# B&R Automation Studio project A2019059_Linka_Power_CP (part 19)

```iecst
            IF NOT SC_P1_Srobovanie.Switch2 AND SC_OvlManipulatora_OsY.Step = 1 AND P1_Srobovacky_VychodziaPozicia AND P1_Srobovanie.STAV.OsX_PoziciaDosiahnuta AND Safety.STAV.P1_ZonaBunky_AKTIVNA THEN
                OsY_POLOHUJ:= TRUE;
                SC_P1_Srobovanie.Switch2:= TRUE;
            END_IF

            IF P1_Srobovanie.STAV.OsX_PoziciaDosiahnuta AND P1_Srobovanie.STAV.OsY_PoziciaDosiahnuta THEN
                P1_Srobovanie.STAV.OsX_PoziciaDosiahnuta:= FALSE;
                P1_Srobovanie.STAV.OsY_PoziciaDosiahnuta:= FALSE;
                SC_P1_Srobovanie.ResetStep:= TRUE;
                SC_P1_Srobovanie.Step:= 503;
            END_IF

        503:
            SC_P1_Srobovanie.StepName:='503 - Inicializacia - zahodenie skrutky K30';
            SC_P1_Srobovanie.IdleTime.PT:= T#30s;
            SC_P1_Srobovanie.AlarmTime.PT:= T#30s;
            SC_P1_Srobovanie.IdleTime.IN:= TRUE;

            IF NOT SC_P1_Srobovanie.Switch1 THEN
                P1_Srobovanie.SkrutkovaciSet_K30.Cistenie:= TRUE;
                SC_P1_Srobovanie.Switch1:= TRUE;
            END_IF

            IF P1_Srobovanie.SkrutkovaciSet_K30.CistenieUkoncene AND P1_Srobovanie.IN.SkrutkK30_ZASUNUTY_MS20 THEN
                P1_Srobovanie.SkrutkovaciSet_K30.Cistenie:= FALSE;
            END_IF

            IF NOT P1_Srobovanie.SkrutkovaciSet_K30.Cistenie AND P1_Srobovanie.SkrutkovaciSet_K30.SkrutkaK30_Pripravena AND SC_P1_Srobovanie.Switch1 THEN
                P1_Srobovanie.STAV.Cistenie_K30_BUSY:= FALSE;
                P1_Srobovanie.RR_SkrutkovackaK30_CISTENIE:= FALSE;
                SC_P1_Srobovanie.ResetStep:= TRUE;
                SC_P1_Srobovanie.Step:= FazaNavratu;
            ELSIF SC_P1_Srobovanie.IdleTime.Q THEN
                SC_P1_Srobovanie.ResetStep:= TRUE;
                SC_P1_Srobovanie.Step:= 505;
            END_IF

        505:
            SC_P1_Srobovanie.StepName:='505 - Inicializacia - cakam na opatovne spustenie cistenia skrutkovacky K30';
            SC_P1_Srobovanie.IdleTime.PT:= T#2s;
            SC_P1_Srobovanie.AlarmTime.PT:= T#30s;

            IF NOT SC_P1_Srobovanie.Switch1 THEN
                P1_Srobovanie.SkrutkovaciSet_K30.Reset:= TRUE;
                P1_Srobovanie.SkrutkovaciSet_K30.Cistenie:= FALSE;
                SC_P1_Srobovanie.IdleTime.IN:= TRUE;
                SC_P1_Srobovanie.Switch1:= TRUE;
            END_IF

            IF SC_P1_Srobovanie.IdleTime.Q THEN
                SC_P1_Srobovanie.ResetStep:= TRUE;
                SC_P1_Srobovanie.Step:= 503;
            END_IF

            //Čistenie skrutkovačky M4//
        510:
            SC_P1_Srobovanie.StepName:='510 - Automaticky Rezim - cistenie skrutkovacky M4';
            SC_P1_Srobovanie.IdleTime.PT:= T#200ms;
            SC_P1_Srobovanie.AlarmTime.PT:= T#5s;

            P1_Srobovanie.PAR.OsX_ZadanaPozicia:= 15; //mm
            P1_Srobovanie.PAR.OsY_ZadanaPozicia:= 157; //mm

            IF NOT SC_P1_Srobovanie.Switch1 AND SC_OvlManipulatora_OsX.Step = 1 AND P1_Srobovacky_VychodziaPozicia AND Safety.STAV.P1_ZonaBunky_AKTIVNA THEN
                P1_Srobovanie.SkrutkovaciSet_M4.SkrutkaM4_Odobrata:= FALSE;
                P1_Srobovanie.SkrutkovaciSet_M4.Automat:= TRUE;
                P1_Srobovanie.SkrutkovaciSet_M4.Reset:= TRUE;
                OsX_POLOHUJ:= TRUE;
                SC_P1_Srobovanie.Switch1:= TRUE;
            END_IF

            IF NOT SC_P1_Srobovanie.Switch2 AND SC_OvlManipulatora_OsY.Step = 1 AND P1_Srobovacky_VychodziaPozicia AND P1_Srobovanie.STAV.OsX_PoziciaDosiahnuta AND Safety.STAV.P1_ZonaBunky_AKTIVNA THEN
                OsY_POLOHUJ:= TRUE;
                SC_P1_Srobovanie.Switch2:= TRUE;
            END_IF

            IF P1_Srobovanie.STAV.OsX_PoziciaDosiahnuta AND P1_Srobovanie.STAV.OsY_PoziciaDosiahnuta THEN
                P1_Srobovanie.STAV.OsX_PoziciaDosiahnuta:= FALSE;
                P1_Srobovanie.STAV.OsY_PoziciaDosiahnuta:= FALSE;
                SC_P1_Srobovanie.ResetStep:= TRUE;
                SC_P1_Srobovanie.Step:= 513;
            END_IF

        513:
            SC_P1_Srobovanie.StepName:='513 - Inicializacia - zahodenie skrutky M4';
            SC_P1_Srobovanie.IdleTime.PT:= T#30s;
            SC_P1_Srobovanie.AlarmTime.PT:= T#30s;
            SC_P1_Srobovanie.IdleTime.IN:= TRUE;

            IF NOT SC_P1_Srobovanie.Switch1 THEN
                P1_Srobovanie.SkrutkovaciSet_M4.Cistenie:= TRUE;
                SC_P1_Srobovanie.Switch1:= TRUE;
            END_IF

            IF P1_Srobovanie.SkrutkovaciSet_M4.CistenieUkoncene AND P1_Srobovanie.IN.SkrutkM4_ZASUNUTY_MS17 THEN
                P1_Srobovanie.SkrutkovaciSet_M4.Cistenie:= FALSE;
            END_IF

            IF NOT P1_Srobovanie.SkrutkovaciSet_M4.Cistenie AND P1_Srobovanie.SkrutkovaciSet_M4.SkrutkaM4_Pripravena AND SC_P1_Srobovanie.Switch1 THEN
                P1_Srobovanie.STAV.Cistenie_M4_BUSY:= FALSE;
                P1_Srobovanie.RR_SkrutkovackaM4_CISTENIE:= FALSE;
                SC_P1_Srobovanie.ResetStep:= TRUE;
                SC_P1_Srobovanie.Step:= FazaNavratu;
            ELSIF SC_P1_Srobovanie.IdleTime.Q THEN
                SC_P1_Srobovanie.ResetStep:= TRUE;
                SC_P1_Srobovanie.Step:= 515;
            END_IF

        515:
            SC_P1_Srobovanie.StepName:='515 - Inicializacia - cakam na opatovne spustenie cistenia skrutkovacky M4';
            SC_P1_Srobovanie.IdleTime.PT:= T#2s;
            SC_P1_Srobovanie.AlarmTime.PT:= T#30s;

            IF NOT SC_P1_Srobovanie.Switch1 THEN
                P1_Srobovanie.SkrutkovaciSet_M4.Reset:= TRUE;
                P1_Srobovanie.SkrutkovaciSet_M4.Cistenie:= FALSE;
                SC_P1_Srobovanie.IdleTime.IN:= TRUE;
                SC_P1_Srobovanie.Switch1:= TRUE;
            END_IF

            IF SC_P1_Srobovanie.IdleTime.Q THEN
                SC_P1_Srobovanie.ResetStep:= TRUE;
                SC_P1_Srobovanie.Step:= 513;
            END_IF

            //*******************************************************Manuálny režim*******************************************************************************//
        700:
            SC_P1_Srobovanie.StepName:='700 - Manualny Rezim';
            SC_P1_Srobovanie.IdleTime.PT:= T#8s;
            SC_P1_Srobovanie.AlarmTime.PT:= T#5s;

            P1_Srobovanie.ServoManipulOsX_M20.PAR.JoggAcceleration:= (P1_Srobovanie.PAR.OsX_JoggRychlost * 10);
            P1_Srobovanie.ServoManipulOsX_M20.PAR.JoggDeceleration:= (P1_Srobovanie.PAR.OsX_JoggRychlost * 10);
            P1_Srobovanie.ServoManipulOsX_M20.PAR.JoggVelocity:= P1_Srobovanie.PAR.OsX_JoggRychlost;
            P1_Srobovanie.ServoManipulOsX_M20.PAR.JoggPoziciaLimitVPRED:= 60.0;
            P1_Srobovanie.ServoManipulOsX_M20.PAR.JoggPoziciaLimitVZAD:= 0.0;
            P1_Srobovanie.ServoManipulOsX_M20.CMD.JoggLimit_ACTIVE:= TRUE;

            P1_Srobovanie.ServoManipulOsY_M19.PAR.JoggAcceleration:= (P1_Srobovanie.PAR.OsY_JoggRychlost * 10);
            P1_Srobovanie.ServoManipulOsY_M19.PAR.JoggDeceleration:= (P1_Srobovanie.PAR.OsY_JoggRychlost * 10);
            P1_Srobovanie.ServoManipulOsY_M19.PAR.JoggVelocity:= P1_Srobovanie.PAR.OsY_JoggRychlost;
            P1_Srobovanie.ServoManipulOsY_M19.PAR.JoggPoziciaLimitVPRED:= 290.0;
            P1_Srobovanie.ServoManipulOsY_M19.PAR.JoggPoziciaLimitVZAD:= 0.0;
            P1_Srobovanie.ServoManipulOsY_M19.CMD.JoggLimit_ACTIVE:= TRUE;

            //Ovládanie vysunutia skrutkovačky M4//
            P1_Srobovanie.OUT.SkrutkM4_VYSUN_YV79:= P1_Srobovanie.RR_SkrutkovackuM4_VYSUN;

            //Ovládanie vysunutia skrutkovačky M5//
            P1_Srobovanie.OUT.SkrutkM5_VYSUN_YV104:= P1_Srobovanie.RR_SkrutkovackuM5_VYSUN;

            //Ovládanie vysunutia skrutkovačky K30//
            P1_Srobovanie.OUT.SkrutkK30_VYSUN_YV89:= P1_Srobovanie.RR_SkrutkovackuK30_VYSUN;

            //Spustenie čistenia skrutkovačiek//
            IF P1_Srobovanie.RR_SkrutkovackaM4_CISTENIE THEN
                P1_Srobovanie.STAV.Cistenie_M4_BUSY:= TRUE;
                FazaNavratu:= 700;
                SC_P1_Srobovanie.ResetStep:= TRUE;
                SC_P1_Srobovanie.Step:= 510;
            ELSIF P1_Srobovanie.RR_SkrutkovackaK30_CISTENIE THEN
                P1_Srobovanie.STAV.Cistenie_K30_BUSY:= TRUE;
                FazaNavratu:= 700;
                SC_P1_Srobovanie.ResetStep:= TRUE;
                SC_P1_Srobovanie.Step:= 500;
            END_IF

            //Prisávanie skrutky M5//
            IF P1_Srobovanie.RR_PrisavanieSkrutkyM5 THEN
                P1_Srobovanie.OUT.SkrutkM5_PrisavSkrut_VYPNI_YV109:= FALSE;
                P1_Srobovanie.OUT.SkrutkM5_PrisavSkrut_ZAPNI_YV105:= TRUE;
            ELSE
                P1_Srobovanie.OUT.SkrutkM5_PrisavSkrut_ZAPNI_YV105:= FALSE;
                P1_Srobovanie.OUT.SkrutkM5_PrisavSkrut_VYPNI_YV109:= TRUE;
            END_IF

            //Polohovanie na pozície skrutiek//
            IF P1_Srobovanie.RR_PolohujNaPoziciuSkrutky_4F THEN
                IF P1_Srobovanie.PAR.RR_IndexPozicieSkrutky_4F = 0 THEN  //Lavá K30
                    SC_P1_Srobovanie.ResetStep:= TRUE;
                    SC_P1_Srobovanie.Step:= 110;
                ELSIF P1_Srobovanie.PAR.RR_IndexPozicieSkrutky_4F = 1 THEN  //Pravá K30
                    SC_P1_Srobovanie.ResetStep:= TRUE;
                    SC_P1_Srobovanie.Step:= 130;
                ELSIF P1_Srobovanie.PAR.RR_IndexPozicieSkrutky_4F = 2 THEN  //Zadná M4
                    SC_P1_Srobovanie.ResetStep:= TRUE;
                    SC_P1_Srobovanie.Step:= 150;
                ELSIF P1_Srobovanie.PAR.RR_IndexPozicieSkrutky_4F = 3 THEN  //Predná M4
                    SC_P1_Srobovanie.ResetStep:= TRUE;
                    SC_P1_Srobovanie.Step:= 170;
                ELSIF P1_Srobovanie.PAR.RR_IndexPozicieSkrutky_4F = 4 THEN  //Stredná M4
                    SC_P1_Srobovanie.ResetStep:= TRUE;
                    SC_P1_Srobovanie.Step:= 190;
                END_IF
            ELSIF P1_Srobovanie.RR_PolohujNaPoziciuSkrutky_5F THEN
                IF P1_Srobovanie.PAR.RR_IndexPozicieSkrutky_5F = 0 THEN  //Lavá K30
                    SC_P1_Srobovanie.ResetStep:= TRUE;
                    SC_P1_Srobovanie.Step:= 200;
                ELSIF P1_Srobovanie.PAR.RR_IndexPozicieSkrutky_5F = 1 THEN  //Pravá K30
                    SC_P1_Srobovanie.ResetStep:= TRUE;
                    SC_P1_Srobovanie.Step:= 220;
                ELSIF P1_Srobovanie.PAR.RR_IndexPozicieSkrutky_5F = 2 THEN  //Zadná M4
                    SC_P1_Srobovanie.ResetStep:= TRUE;
                    SC_P1_Srobovanie.Step:= 240;
                ELSIF P1_Srobovanie.PAR.RR_IndexPozicieSkrutky_5F = 3 THEN  //Predná M4
                    SC_P1_Srobovanie.ResetStep:= TRUE;
                    SC_P1_Srobovanie.Step:= 260;
                ELSIF P1_Srobovanie.PAR.RR_IndexPozicieSkrutky_5F = 4 THEN  //Stredná M4
                    SC_P1_Srobovanie.ResetStep:= TRUE;
                    SC_P1_Srobovanie.Step:= 280;
                END_IF
            ELSIF  P1_Srobovanie.RR_PolohujNaPoziciuSkrutky_5H THEN
                IF P1_Srobovanie.PAR.RR_IndexPozicieSkrutky_5H = 0 THEN  //Lavá K30
                    SC_P1_Srobovanie.ResetStep:= TRUE;
                    SC_P1_Srobovanie.Step:= 300;
                ELSIF P1_Srobovanie.PAR.RR_IndexPozicieSkrutky_5H = 1 THEN  //Pravá K30
                    SC_P1_Srobovanie.ResetStep:= TRUE;
                    SC_P1_Srobovanie.Step:= 320;
                ELSIF P1_Srobovanie.PAR.RR_IndexPozicieSkrutky_5H = 2 THEN  //Lavá M5
                    SC_P1_Srobovanie.ResetStep:= TRUE;
                    SC_P1_Srobovanie.Step:= 346;
                ELSIF P1_Srobovanie.PAR.RR_IndexPozicieSkrutky_5H = 3 THEN  //Pravá M5
                    SC_P1_Srobovanie.ResetStep:= TRUE;
                    SC_P1_Srobovanie.Step:= 366;
                ELSIF P1_Srobovanie.PAR.RR_IndexPozicieSkrutky_5H = 4 THEN  //Stredná M4
                    SC_P1_Srobovanie.ResetStep:= TRUE;
                    SC_P1_Srobovanie.Step:= 386;
                ELSIF P1_Srobovanie.PAR.RR_IndexPozicieSkrutky_5H = 5 THEN  //Pozícia odobratia skrutky M5
                    SC_P1_Srobovanie.ResetStep:= TRUE;
                    SC_P1_Srobovanie.Step:= 340;
                END_IF
            END_IF

    END_CASE

END_PROGRAM

PROGRAM _EXIT
	(* Insert code here *)

END_PROGRAM
```

#### Variables.var - Local variables
```iecst
VAR
	SC_OvlManipulatora_OsX : SequenceControlTyp;
	OsX_JoggVPRED : BOOL;
	OsX_JoggVZAD : BOOL;
	OsX_POLOHUJ : BOOL;
	OsX_HOME : BOOL;
	OsX_STOP : BOOL;
	SC_OvlManipulatora_OsY : SequenceControlTyp;
	OsY_JoggVPRED : BOOL;
	OsY_JoggVZAD : BOOL;
	OsY_POLOHUJ : BOOL;
	OsY_HOME : BOOL;
	OsY_STOP : BOOL;
	ZadanaPoziciaUINT_OsX : UINT;
	AktualnaPoziciaUINT_OsX : UINT;
	ZadanaPoziciaUINT_OsY : UINT;
	AktualnaPoziciaUINT_OsY : UINT;
	Start : BOOL;
	TEST : BOOL;
	Triger_0 : BOOL;
	CasPowerON_OsY : TON;
	CasPowerON_OsX : TON;
	i : USINT;
	CasSrobovania : REAL;
	K30_Moment_ToleranciaMAX_REAL : REAL;
	K30_Moment_ToleranciaMIN_REAL : REAL;
	K30_DosiahnutyMoment_REAL : REAL;
	M5_DosiahnutyMoment_REAL : REAL;
	M5_Moment_ToleranciaMAX_REAL : REAL;
	M5_Moment_ToleranciaMIN_REAL : REAL;
	M4_DosiahnutyMoment_REAL : REAL;
	M4_Moment_ToleranciaMAX_REAL : REAL;
	M4_Moment_ToleranciaMIN_REAL : REAL;
	K30_PrevodMomentu : PrevodMomentu;
	M4_PrevodMomentu : PrevodMomentu;
	M5_PrevodMomentu : PrevodMomentu;
	CasZastaveniaServa : TON;
	CasZastaveniaServa_2 : TON;
	FazaNavratu : UINT;
	CasKontrolyZasobSkrutiek_K30 : TON;
	CasKontrolyZasobSkrutiek_M5 : TON;
	CasKontrolyZasobSkrutiek_M4 : TON;
END_VAR
(******Zápis do ParID serva*************)
VAR
	MC_BR_ProcessParID_AcpAx_0 : MC_BR_ProcessParID_AcpAx := (0);
	McAcpAxProcessParIDType_0 : ARRAY[0..1] OF McAcpAxProcessParIDType;
	OsX_NovaHodnotaMomentu_POS : REAL := 0.0;
	OsX_NovaHodnotaMomentu_NEG : REAL := 0.0;
	MC_BR_ProcessParID_AcpAx_1 : MC_BR_ProcessParID_AcpAx := (0);
	McAcpAxProcessParIDType_1 : ARRAY[0..1] OF McAcpAxProcessParIDType;
	OsY_NovaHodnotaMomentu_POS : REAL := 0.0;
	OsY_NovaHodnotaMomentu_NEG : REAL := 0.0;
END_VAR
```

#### OvlManipulatora_OsX.st
```iecst
ACTION OvlManipulatora_OsX:

	//*****************************Axis 7************************************//
	//Otáčka serva = 10mm//
	//Motor má absolútny encodér//

    //ENABLE knižnice//
    IF P1_Srobovanie.ServoManipulOsX_M20.STATUS.Communication_READY THEN
        P1_Srobovanie.ServoManipulOsX_M20.CMD.ENABLE:= TRUE;
    ELSE
        P1_Srobovanie.ServoManipulOsX_M20.CMD.ENABLE:= FALSE;
    END_IF

	//Zapnutie serva//
	CasPowerON_OsX.IN:= P1_Srobovanie.ServoManipulOsX_M20.STATUS.ReadyToPower_ON AND P1_Srobovanie.STAV.OsX_LimitSnimace_BUSY AND P1_Srobovanie.ServoManipulOsX_M20.STATUS.EnableSwitch_ACTIVE AND NOT P1_Srobovanie.ServoManipulOsX_M20.STATUS.ERROR;
	IF CasPowerON_OsX.Q THEN
		P1_Srobovanie.ServoManipulOsX_M20.CMD.POWER:= TRUE;
	ELSE
		P1_Srobovanie.ServoManipulOsX_M20.CMD.POWER:= FALSE;
	END_IF

	CasPowerON_OsX.PT:= T#1s;
	CasPowerON_OsX();

    //Zobrazenie stavou a parametrov serva//
    P1_Srobovanie.STAV.OsX_AktualnaPozicia:= P1_Srobovanie.ServoManipulOsX_M20.STATUS.ActualPosition;
    P1_Srobovanie.STAV.OsX_AktualnaRychlost:= P1_Srobovanie.ServoManipulOsX_M20.STATUS.ActualVelocity;
	P1_Srobovanie.STAV.OsX_AktualnyMoment:= P1_Srobovanie.ServoManipulOsX_M20.STATUS.ActualTorque;
	P1_Srobovanie.STAV.OsX_HomingOK:= P1_Srobovanie.ServoManipulOsX_M20.STATUS.Homing_OK;
	P1_Srobovanie.STAV.OsX_BUSY:= P1_Srobovanie.ServoManipulOsX_M20.STATUS.MoveAbsolute_BUSY;
	P1_Srobovanie.STAV.OsX_JoggLimitDosiahnuty:= P1_Srobovanie.ServoManipulOsX_M20.STATUS.JoggLimit_Dosiahnuty;

	//Zadané parametre serva//
	P1_Srobovanie.ServoManipulOsX_M20.HomePAR.Acceleration:= 50;
	P1_Srobovanie.ServoManipulOsX_M20.HomePAR.HomingVelocity:= 5;
	P1_Srobovanie.ServoManipulOsX_M20.HomePAR.StartVelocity:= 10;
	P1_Srobovanie.ServoManipulOsX_M20.HomePAR.Position:= -29045.2;    //Offset homing pozície pre absolutny snímač
	P1_Srobovanie.ServoManipulOsX_M20.HomePAR.HomingMode:= 3; //0 - direct, 1- refrenčný snímač, 2 - limitný snímač, 3 - absolutny encoder, 4 - na moment//

	P1_Srobovanie.ServoManipulOsX_M20.PAR.Acceleration:= P1_RemPremenne.P1_ManipSrob_OsX_Rychlost*10;
	P1_Srobovanie.ServoManipulOsX_M20.PAR.Deceleration:= P1_RemPremenne.P1_ManipSrob_OsX_Rychlost*10;
	P1_Srobovanie.ServoManipulOsX_M20.PAR.StopDeceleration:= P1_RemPremenne.P1_ManipSrob_OsX_Rychlost*10;
	P1_Srobovanie.ServoManipulOsX_M20.PAR.Velocity:= P1_RemPremenne.P1_ManipSrob_OsX_Rychlost;
	P1_Srobovanie.ServoManipulOsX_M20.PAR.Position:= P1_Srobovanie.PAR.OsX_ZadanaPozicia;

	//Zastavenie pohybu serva//
	IF OsX_STOP THEN
		P1_Srobovanie.ServoManipulOsX_M20.CMD.STOP:= TRUE;
		SC_OvlManipulatora_OsX.Step:= 0;
		CasZastaveniaServa_2.IN:= TRUE;
		OsX_STOP:= FALSE;
	END_IF

	IF CasZastaveniaServa_2.Q  THEN
		P1_Srobovanie.ServoManipulOsX_M20.CMD.STOP:= FALSE;
		CasZastaveniaServa_2.IN:= FALSE;
	END_IF

	CasZastaveniaServa_2.PT:= T#2s;
	CasZastaveniaServa_2();

	//Volanie funkcie SequenceControl//
	SequenceControl(SC:= SC_OvlManipulatora_OsX);

	CASE SC_OvlManipulatora_OsX.Step OF

		0:
			SC_OvlManipulatora_OsX.StepName:= '0 - Nulovanie';
			OsX_JoggVPRED:= FALSE;
			OsX_JoggVZAD:= FALSE;
			OsX_POLOHUJ:= FALSE;
			OsX_HOME:= FALSE;
			P1_Srobovanie.ServoManipulOsX_M20.CMD.HOME:= FALSE;
			P1_Srobovanie.ServoManipulOsX_M20.CMD.JoggVPRED:= FALSE;
			P1_Srobovanie.ServoManipulOsX_M20.CMD.JoggVZAD:= FALSE;
			P1_Srobovanie.ServoManipulOsX_M20.CMD.MoveAbsolute:= FALSE;

			IF SC_P1_Srobovanie.Step <> 0 AND P1_Srobovanie.ServoManipulOsX_M20.STATUS.Power_ON AND NOT P1_Srobovanie.ServoManipulOsX_M20.STATUS.ERROR AND NOT P1_Srobovanie.ServoManipulOsX_M20.STATUS.STOP_ACTIVE THEN
				SC_OvlManipulatora_OsX.ResetStep:= TRUE;
				SC_OvlManipulatora_OsX.Step:= 1;
			END_IF

		1:
			SC_OvlManipulatora_OsX.StepName:= '1 - Rozhodnutie o cinnosti';
			IF OsX_JoggVPRED THEN
				SC_OvlManipulatora_OsX.Step:= 10;
			ELSIF OsX_JoggVZAD THEN
				SC_OvlManipulatora_OsX.Step:= 20;
			ELSIF OsX_HOME THEN
				SC_OvlManipulatora_OsX.Step:= 30;
			ELSIF OsX_POLOHUJ THEN
				SC_OvlManipulatora_OsX.Step:= 40;
			END_IF

		10:
			SC_OvlManipulatora_OsX.StepName:= '10 - Jogg VPRED';
			SC_OvlManipulatora_OsX.IdleTime.PT:= T#3s;
			SC_OvlManipulatora_OsX.AlarmTime.PT:= T#3s;

			IF NOT SC_OvlManipulatora_OsX.Switch1 THEN
				P1_Srobovanie.ServoManipulOsX_M20.CMD.JoggVPRED:= TRUE;
				SC_OvlManipulatora_OsX.Switch1:= TRUE;
			END_IF

			IF NOT OsX_JoggVPRED THEN
				SC_OvlManipulatora_OsX.ResetStep:= TRUE;
				SC_OvlManipulatora_OsX.Step:= 0;
			END_IF

		20:
			SC_OvlManipulatora_OsX.StepName:= '20 - Jogg VZAD';
			SC_OvlManipulatora_OsX.IdleTime.PT:= T#3s;
			SC_OvlManipulatora_OsX.AlarmTime.PT:= T#3s;

			IF NOT SC_OvlManipulatora_OsX.Switch1 THEN
				P1_Srobovanie.ServoManipulOsX_M20.CMD.JoggVZAD:= TRUE;
				SC_OvlManipulatora_OsX.Switch1:= TRUE;
			END_IF

			IF NOT OsX_JoggVZAD THEN
				SC_OvlManipulatora_OsX.ResetStep:= TRUE;
				SC_OvlManipulatora_OsX.Step:= 0;
			END_IF

		30:
			SC_OvlManipulatora_OsX.StepName:= '30 - Homing';
			SC_OvlManipulatora_OsX.IdleTime.PT:= T#500ms;
			SC_OvlManipulatora_OsX.AlarmTime.PT:= T#3s;

			IF NOT SC_OvlManipulatora_OsX.Switch1 THEN
				P1_Srobovanie.ServoManipulOsX_M20.CMD.HOME:= TRUE;
				SC_OvlManipulatora_OsX.IdleTime.IN:= TRUE;
				SC_OvlManipulatora_OsX.Switch1:= TRUE;
			END_IF

			IF P1_Srobovanie.ServoManipulOsX_M20.STATUS.Homing_OK AND SC_OvlManipulatora_OsX.IdleTime.Q THEN
				SC_OvlManipulatora_OsX.ResetStep:= TRUE;
				SC_OvlManipulatora_OsX.Step:= 0;
			END_IF

		40:
			SC_OvlManipulatora_OsX.StepName:= '40 - Polohovanie';
			SC_OvlManipulatora_OsX.IdleTime.PT:= T#500ms;
			SC_OvlManipulatora_OsX.AlarmTime.PT:= T#3s;

			ZadanaPoziciaUINT_OsX:= LREAL_TO_UINT(P1_Srobovanie.PAR.OsX_ZadanaPozicia);
			AktualnaPoziciaUINT_OsX:= LREAL_TO_UINT(P1_Srobovanie.STAV.OsX_AktualnaPozicia);

			IF NOT SC_OvlManipulatora_OsX.Switch1 THEN
				P1_Srobovanie.ServoManipulOsX_M20.CMD.MoveAbsolute:= TRUE;
				SC_OvlManipulatora_OsX.Switch1:= TRUE;
			END_IF

			IF (AktualnaPoziciaUINT_OsX = ZadanaPoziciaUINT_OsX) AND P1_Srobovanie.ServoManipulOsX_M20.STATUS.MoveAbsolute_DONE THEN
				P1_Srobovanie.STAV.OsX_PoziciaDosiahnuta:= TRUE;
				SC_OvlManipulatora_OsX.ResetStep:= TRUE;
				SC_OvlManipulatora_OsX.Step:= 0;
			END_IF

	END_CASE

END_ACTION
```

#### OvlManipulatora_OsY.st
```iecst
ACTION OvlManipulatora_OsY:

	//************************Axis 8*******************************//
	//Otáčka serva = 10mm//
	//Motor má absolútny encodér//

    //ENABLE knižnice//
    IF P1_Srobovanie.ServoManipulOsY_M19.STATUS.Communication_READY THEN
        P1_Srobovanie.ServoManipulOsY_M19.CMD.ENABLE:= TRUE;
    ELSE
        P1_Srobovanie.ServoManipulOsY_M19.CMD.ENABLE:= FALSE;
    END_IF

	//Zapnutie serva//
	CasPowerON_OsY.IN:= P1_Srobovanie.ServoManipulOsY_M19.STATUS.ReadyToPower_ON AND P1_Srobovanie.STAV.OsY_LimitSnimace_BUSY AND P1_Srobovanie.ServoManipulOsY_M19.STATUS.EnableSwitch_ACTIVE AND NOT P1_Srobovanie.ServoManipulOsY_M19.STATUS.ERROR;
	IF CasPowerON_OsY.Q THEN
		P1_Srobovanie.ServoManipulOsY_M19.CMD.POWER:= TRUE;
	ELSE
		P1_Srobovanie.ServoManipulOsY_M19.CMD.POWER:= FALSE;
	END_IF

	CasPowerON_OsY.PT:= T#1s;
	CasPowerON_OsY();

	//Zobrazenie stavou a parametrov serva//
	P1_Srobovanie.STAV.OsY_AktualnaPozicia:= P1_Srobovanie.ServoManipulOsY_M19.STATUS.ActualPosition;
	P1_Srobovanie.STAV.OsY_AktualnaRychlost:= P1_Srobovanie.ServoManipulOsY_M19.STATUS.ActualVelocity;
	P1_Srobovanie.STAV.OsY_AktualnyMoment:= P1_Srobovanie.ServoManipulOsY_M19.STATUS.ActualTorque;
	P1_Srobovanie.STAV.OsY_HomingOK:= P1_Srobovanie.ServoManipulOsY_M19.STATUS.Homing_OK;
	P1_Srobovanie.STAV.OsY_BUSY:= P1_Srobovanie.ServoManipulOsY_M19.STATUS.MoveAbsolute_BUSY;
	P1_Srobovanie.STAV.OsY_JoggLimitDosiahnuty:= P1_Srobovanie.ServoManipulOsY_M19.STATUS.JoggLimit_Dosiahnuty;

	//Zadané parametre serva//
	P1_Srobovanie.ServoManipulOsY_M19.HomePAR.Acceleration:= 50;
	P1_Srobovanie.ServoManipulOsY_M19.HomePAR.HomingVelocity:= 5;
	P1_Srobovanie.ServoManipulOsY_M19.HomePAR.StartVelocity:= 10;
	P1_Srobovanie.ServoManipulOsY_M19.HomePAR.Position:= -27941.0;    //Offset homing pozície pre absolutny snímač
	P1_Srobovanie.ServoManipulOsY_M19.HomePAR.HomingMode:= 3; //0 - direct, 1- refrenčný snímač, 2 - limitný snímač, 3 - absolutny encoder, 4 - na moment//

	P1_Srobovanie.ServoManipulOsY_M19.PAR.Acceleration:= P1_RemPremenne.P1_ManipSrob_OsY_Rychlost*10;
	P1_Srobovanie.ServoManipulOsY_M19.PAR.Deceleration:= P1_RemPremenne.P1_ManipSrob_OsY_Rychlost*10;
	P1_Srobovanie.ServoManipulOsY_M19.PAR.StopDeceleration:= P1_RemPremenne.P1_ManipSrob_OsY_Rychlost*10;
	P1_Srobovanie.ServoManipulOsY_M19.PAR.Velocity:= P1_RemPremenne.P1_ManipSrob_OsY_Rychlost;
	P1_Srobovanie.ServoManipulOsY_M19.PAR.Position:= P1_Srobovanie.PAR.OsY_ZadanaPozicia;

	//Zastavenie pohybu serva//
	IF OsY_STOP THEN
		P1_Srobovanie.ServoManipulOsY_M19.CMD.STOP:= TRUE;
		SC_OvlManipulatora_OsY.Step:= 0;
		CasZastaveniaServa.IN:= TRUE;
		OsY_STOP:= FALSE;
	END_IF

	IF CasZastaveniaServa.Q THEN
		P1_Srobovanie.ServoManipulOsY_M19.CMD.STOP:= FALSE;
		CasZastaveniaServa.IN:= FALSE;
	END_IF

	CasZastaveniaServa.PT:= T#2s;
	CasZastaveniaServa();

	//Volanie funkcie SequenceControl//
	SequenceControl(SC:= SC_OvlManipulatora_OsY);

	CASE SC_OvlManipulatora_OsY.Step OF

		0:
			SC_OvlManipulatora_OsY.StepName:= '0 - Nulovanie';
			OsY_JoggVPRED:= FALSE;
			OsY_JoggVZAD:= FALSE;
			OsY_POLOHUJ:= FALSE;
			OsY_HOME:= FALSE;
			P1_Srobovanie.ServoManipulOsY_M19.CMD.HOME:= FALSE;
			P1_Srobovanie.ServoManipulOsY_M19.CMD.JoggVPRED:= FALSE;
			P1_Srobovanie.ServoManipulOsY_M19.CMD.JoggVZAD:= FALSE;
			P1_Srobovanie.ServoManipulOsY_M19.CMD.MoveAbsolute:= FALSE;

			IF SC_P1_Srobovanie.Step <> 0 AND P1_Srobovanie.ServoManipulOsY_M19.STATUS.Power_ON AND NOT P1_Srobovanie.ServoManipulOsY_M19.STATUS.ERROR AND NOT P1_Srobovanie.ServoManipulOsY_M19.STATUS.STOP_ACTIVE THEN
				SC_OvlManipulatora_OsY.ResetStep:= TRUE;
				SC_OvlManipulatora_OsY.Step:= 1;
			END_IF

		1:
			SC_OvlManipulatora_OsY.StepName:= '1 - Rozhodnutie o cinnosti';
			IF OsY_JoggVPRED THEN
				SC_OvlManipulatora_OsY.Step:= 10;
			ELSIF OsY_JoggVZAD THEN
				SC_OvlManipulatora_OsY.Step:= 20;
			ELSIF OsY_HOME THEN
				SC_OvlManipulatora_OsY.Step:= 30;
			ELSIF OsY_POLOHUJ THEN
				SC_OvlManipulatora_OsY.Step:= 40;
			END_IF

		10:
			SC_OvlManipulatora_OsY.StepName:= '10 - Jogg VPRED';
			SC_OvlManipulatora_OsY.IdleTime.PT:= T#3s;
			SC_OvlManipulatora_OsY.AlarmTime.PT:= T#3s;

			IF NOT SC_OvlManipulatora_OsY.Switch1 THEN
				P1_Srobovanie.ServoManipulOsY_M19.CMD.JoggVPRED:= TRUE;
				SC_OvlManipulatora_OsY.Switch1:= TRUE;
			END_IF

			IF NOT OsY_JoggVPRED THEN
				SC_OvlManipulatora_OsY.ResetStep:= TRUE;
				SC_OvlManipulatora_OsY.Step:= 0;
			END_IF

		20:
			SC_OvlManipulatora_OsY.StepName:= '20 - Jogg VZAD';
			SC_OvlManipulatora_OsY.IdleTime.PT:= T#3s;
			SC_OvlManipulatora_OsY.AlarmTime.PT:= T#3s;

			IF NOT SC_OvlManipulatora_OsY.Switch1 THEN
				P1_Srobovanie.ServoManipulOsY_M19.CMD.JoggVZAD:= TRUE;
				SC_OvlManipulatora_OsY.Switch1:= TRUE;
			END_IF

			IF NOT OsY_JoggVZAD THEN
				SC_OvlManipulatora_OsY.ResetStep:= TRUE;
				SC_OvlManipulatora_OsY.Step:= 0;
			END_IF

		30:
			SC_OvlManipulatora_OsY.StepName:= '30 - Homing';
			SC_OvlManipulatora_OsY.IdleTime.PT:= T#500ms;
			SC_OvlManipulatora_OsY.AlarmTime.PT:= T#3s;

			IF NOT SC_OvlManipulatora_OsY.Switch1 THEN
				P1_Srobovanie.ServoManipulOsY_M19.CMD.HOME:= TRUE;
				SC_OvlManipulatora_OsY.IdleTime.IN:= TRUE;
				SC_OvlManipulatora_OsY.Switch1:= TRUE;
			END_IF

			IF P1_Srobovanie.ServoManipulOsY_M19.STATUS.Homing_OK AND SC_OvlManipulatora_OsY.IdleTime.Q THEN
				SC_OvlManipulatora_OsY.ResetStep:= TRUE;
				SC_OvlManipulatora_OsY.Step:= 0;
			END_IF

		40:
			SC_OvlManipulatora_OsY.StepName:= '40 - Polohovanie';
			SC_OvlManipulatora_OsY.IdleTime.PT:= T#500ms;
			SC_OvlManipulatora_OsY.AlarmTime.PT:= T#3s;

			ZadanaPoziciaUINT_OsY:= LREAL_TO_UINT(P1_Srobovanie.PAR.OsY_ZadanaPozicia);
			AktualnaPoziciaUINT_OsY:= LREAL_TO_UINT(P1_Srobovanie.STAV.OsY_AktualnaPozicia);

			IF NOT SC_OvlManipulatora_OsY.Switch1 THEN
				P1_Srobovanie.ServoManipulOsY_M19.CMD.MoveAbsolute:= TRUE;
				SC_OvlManipulatora_OsY.Switch1:= TRUE;
			END_IF

			IF (AktualnaPoziciaUINT_OsY = ZadanaPoziciaUINT_OsY) AND P1_Srobovanie.ServoManipulOsY_M19.STATUS.MoveAbsolute_DONE THEN
				P1_Srobovanie.STAV.OsY_PoziciaDosiahnuta:= TRUE;
				SC_OvlManipulatora_OsY.ResetStep:= TRUE;
				SC_OvlManipulatora_OsY.Step:= 0;
			END_IF

	END_CASE

END_ACTION
```

#### AtlasCopcoKomunikacia.st
```iecst
ACTION AtlasCopcoKomunikacia:

    M4_PrevodMomentu();
    M5_PrevodMomentu();
	K30_PrevodMomentu();
	//*********************************************************Skrutkovacka M5********************************************************************************//
	//Vstupy z AtlasCopco do PLC//
    P1_Srobovanie.Skrutkovacka_M5.Stav_VysledokPotvrdeny:= P1_Srobovanie.PAR.M5_AtlasCopcoInputs[0].0;
    P1_Srobovanie.Skrutkovacka_M5.Stav_EmergencyStop:= P1_Srobovanie.PAR.M5_AtlasCopcoInputs[0].1;
    P1_Srobovanie.Skrutkovacka_M5.Stav_READY_to_START:= P1_Srobovanie.PAR.M5_AtlasCopcoInputs[0].2;
    P1_Srobovanie.Skrutkovacka_M5.Stav_MANUAL:= P1_Srobovanie.PAR.M5_AtlasCopcoInputs[0].3;
    P1_Srobovanie.Skrutkovacka_M5.Stav_UtahovanieUkoncene:= P1_Srobovanie.PAR.M5_AtlasCopcoInputs[0].4;
    P1_Srobovanie.Skrutkovacka_M5.Stav_VysledokUtahovania_NG:= P1_Srobovanie.PAR.M5_AtlasCopcoInputs[0].5;
    P1_Srobovanie.Skrutkovacka_M5.Stav_VysledokUtahovania_OK:= P1_Srobovanie.PAR.M5_AtlasCopcoInputs[0].6;
    P1_Srobovanie.Skrutkovacka_M5.Stav_SmerOtacania_VPRED:= P1_Srobovanie.PAR.M5_AtlasCopcoInputs[0].7;
    P1_Srobovanie.Skrutkovacka_M5.Stav_BUSY:= P1_Srobovanie.PAR.M5_AtlasCopcoInputs[0].8;
    P1_Srobovanie.Skrutkovacka_M5.Stav_ControlerSwitch_ON:= P1_Srobovanie.PAR.M5_AtlasCopcoInputs[0].9;
    P1_Srobovanie.Skrutkovacka_M5.Stav_Station_READY:= P1_Srobovanie.PAR.M5_AtlasCopcoInputs[0].10;
    P1_Srobovanie.Skrutkovacka_M5.Stav_NastrojPripojeny:= P1_Srobovanie.PAR.M5_AtlasCopcoInputs[0].11;
    P1_Srobovanie.Skrutkovacka_M5.Stav_NastrojUtahuje:= P1_Srobovanie.PAR.M5_AtlasCopcoInputs[0].12;

    //Výstupy z PLC do AtlasCopco//
    P1_Srobovanie.PAR.M5_AllasCopcoOutputs[0].0:= P1_Srobovanie.Skrutkovacka_M5.RESET_Poruchy;
    P1_Srobovanie.PAR.M5_AllasCopcoOutputs[0].1:= P1_Srobovanie.Skrutkovacka_M5.RESET_Vysledkov;
    P1_Srobovanie.PAR.M5_AllasCopcoOutputs[0].2:= P1_Srobovanie.Skrutkovacka_M5.START_Skrutkovania;
    P1_Srobovanie.PAR.M5_AllasCopcoOutputs[0].3:= P1_Srobovanie.Skrutkovacka_M5.START_Utahovania;

    //Číslo zadaného programu//
    P1_Srobovanie.PAR.M5_AllasCopcoOutputs[0].16:= P1_Srobovanie.Skrutkovacka_M5.CisloZadanehoProgramu.0;
    P1_Srobovanie.PAR.M5_AllasCopcoOutputs[0].17:= P1_Srobovanie.Skrutkovacka_M5.CisloZadanehoProgramu.1;
    P1_Srobovanie.PAR.M5_AllasCopcoOutputs[0].18:= P1_Srobovanie.Skrutkovacka_M5.CisloZadanehoProgramu.2;
    P1_Srobovanie.PAR.M5_AllasCopcoOutputs[0].19:= P1_Srobovanie.Skrutkovacka_M5.CisloZadanehoProgramu.3;
    P1_Srobovanie.PAR.M5_AllasCopcoOutputs[0].20:= P1_Srobovanie.Skrutkovacka_M5.CisloZadanehoProgramu.4;
    P1_Srobovanie.PAR.M5_AllasCopcoOutputs[0].21:= P1_Srobovanie.Skrutkovacka_M5.CisloZadanehoProgramu.5;
    P1_Srobovanie.PAR.M5_AllasCopcoOutputs[0].22:= P1_Srobovanie.Skrutkovacka_M5.CisloZadanehoProgramu.6;
    P1_Srobovanie.PAR.M5_AllasCopcoOutputs[0].23:= P1_Srobovanie.Skrutkovacka_M5.CisloZadanehoProgramu.7;

    //Číslo aktuálneho programu//
    P1_Srobovanie.Skrutkovacka_M5.Stav_CisloAktualnehoProgramu.0:= P1_Srobovanie.PAR.M5_AtlasCopcoInputs[5].8;
    P1_Srobovanie.Skrutkovacka_M5.Stav_CisloAktualnehoProgramu.1:= P1_Srobovanie.PAR.M5_AtlasCopcoInputs[5].9;
    P1_Srobovanie.Skrutkovacka_M5.Stav_CisloAktualnehoProgramu.2:= P1_Srobovanie.PAR.M5_AtlasCopcoInputs[5].10;
    P1_Srobovanie.Skrutkovacka_M5.Stav_CisloAktualnehoProgramu.3:= P1_Srobovanie.PAR.M5_AtlasCopcoInputs[5].11;
    P1_Srobovanie.Skrutkovacka_M5.Stav_CisloAktualnehoProgramu.4:= P1_Srobovanie.PAR.M5_AtlasCopcoInputs[5].12;
    P1_Srobovanie.Skrutkovacka_M5.Stav_CisloAktualnehoProgramu.5:= P1_Srobovanie.PAR.M5_AtlasCopcoInputs[5].13;
    P1_Srobovanie.Skrutkovacka_M5.Stav_CisloAktualnehoProgramu.6:= P1_Srobovanie.PAR.M5_AtlasCopcoInputs[5].14;
    P1_Srobovanie.Skrutkovacka_M5.Stav_CisloAktualnehoProgramu.7:= P1_Srobovanie.PAR.M5_AtlasCopcoInputs[5].15;

    //Program č.1 - skrutkovanie do plastu
    //Program č.2 - skrutkovanie do kovu

    //Dosiahnutý moment//
//    P1_Srobovanie.STAV.M5_DosiahnutyMoment.0:= P1_Srobovanie.PAR.M5_AtlasCopcoInputs[1].24;
//    P1_Srobovanie.STAV.M5_DosiahnutyMoment.1:= P1_Srobovanie.PAR.M5_AtlasCopcoInputs[1].25;
//    P1_Srobovanie.STAV.M5_DosiahnutyMoment.2:= P1_Srobovanie.PAR.M5_AtlasCopcoInputs[1].26;
//    P1_Srobovanie.STAV.M5_DosiahnutyMoment.3:= P1_Srobovanie.PAR.M5_AtlasCopcoInputs[1].27;
//    P1_Srobovanie.STAV.M5_DosiahnutyMoment.4:= P1_Srobovanie.PAR.M5_AtlasCopcoInputs[1].28;
//    P1_Srobovanie.STAV.M5_DosiahnutyMoment.5:= P1_Srobovanie.PAR.M5_AtlasCopcoInputs[1].29;
//    P1_Srobovanie.STAV.M5_DosiahnutyMoment.6:= P1_Srobovanie.PAR.M5_AtlasCopcoInputs[1].30;
//    P1_Srobovanie.STAV.M5_DosiahnutyMoment.7:= P1_Srobovanie.PAR.M5_AtlasCopcoInputs[1].31;
//    P1_Srobovanie.STAV.M5_DosiahnutyMoment.8:= P1_Srobovanie.PAR.M5_AtlasCopcoInputs[1].16;
//    P1_Srobovanie.STAV.M5_DosiahnutyMoment.9:= P1_Srobovanie.PAR.M5_AtlasCopcoInputs[1].17;
//    P1_Srobovanie.STAV.M5_DosiahnutyMoment.10:= P1_Srobovanie.PAR.M5_AtlasCopcoInputs[1].18;
//    P1_Srobovanie.STAV.M5_DosiahnutyMoment.11:= P1_Srobovanie.PAR.M5_AtlasCopcoInputs[1].19;
//    P1_Srobovanie.STAV.M5_DosiahnutyMoment.12:= P1_Srobovanie.PAR.M5_AtlasCopcoInputs[1].20;
//    P1_Srobovanie.STAV.M5_DosiahnutyMoment.13:= P1_Srobovanie.PAR.M5_AtlasCopcoInputs[1].21;
//    P1_Srobovanie.STAV.M5_DosiahnutyMoment.14:= P1_Srobovanie.PAR.M5_AtlasCopcoInputs[1].22;
//    P1_Srobovanie.STAV.M5_DosiahnutyMoment.15:= P1_Srobovanie.PAR.M5_AtlasCopcoInputs[1].23;
//    P1_Srobovanie.STAV.M5_DosiahnutyMoment.16:= P1_Srobovanie.PAR.M5_AtlasCopcoInputs[1].8;
//    P1_Srobovanie.STAV.M5_DosiahnutyMoment.17:= P1_Srobovanie.PAR.M5_AtlasCopcoInputs[1].9;
//    P1_Srobovanie.STAV.M5_DosiahnutyMoment.18:= P1_Srobovanie.PAR.M5_AtlasCopcoInputs[1].10;
//    P1_Srobovanie.STAV.M5_DosiahnutyMoment.19:= P1_Srobovanie.PAR.M5_AtlasCopcoInputs[1].11;
//    P1_Srobovanie.STAV.M5_DosiahnutyMoment.20:= P1_Srobovanie.PAR.M5_AtlasCopcoInputs[1].12;
//    P1_Srobovanie.STAV.M5_DosiahnutyMoment.21:= P1_Srobovanie.PAR.M5_AtlasCopcoInputs[1].13;
//    P1_Srobovanie.STAV.M5_DosiahnutyMoment.22:= P1_Srobovanie.PAR.M5_AtlasCopcoInputs[1].14;
//    P1_Srobovanie.STAV.M5_DosiahnutyMoment.23:= P1_Srobovanie.PAR.M5_AtlasCopcoInputs[1].15;
//    P1_Srobovanie.STAV.M5_DosiahnutyMoment.24:= P1_Srobovanie.PAR.M5_AtlasCopcoInputs[1].0;
//    P1_Srobovanie.STAV.M5_DosiahnutyMoment.25:= P1_Srobovanie.PAR.M5_AtlasCopcoInputs[1].1;
//    P1_Srobovanie.STAV.M5_DosiahnutyMoment.26:= P1_Srobovanie.PAR.M5_AtlasCopcoInputs[1].2;
//    P1_Srobovanie.STAV.M5_DosiahnutyMoment.27:= P1_Srobovanie.PAR.M5_AtlasCopcoInputs[1].3;
//    P1_Srobovanie.STAV.M5_DosiahnutyMoment.28:= P1_Srobovanie.PAR.M5_AtlasCopcoInputs[1].4;
//    P1_Srobovanie.STAV.M5_DosiahnutyMoment.29:= P1_Srobovanie.PAR.M5_AtlasCopcoInputs[1].5;
//    P1_Srobovanie.STAV.M5_DosiahnutyMoment.30:= P1_Srobovanie.PAR.M5_AtlasCopcoInputs[1].6;
//    P1_Srobovanie.STAV.M5_DosiahnutyMoment.31:= P1_Srobovanie.PAR.M5_AtlasCopcoInputs[1].7;
//    M5_DosiahnutyMoment_REAL:= UDINT_TO_REAL(P1_Srobovanie.STAV.M5_DosiahnutyMoment);
//    IF M5_DosiahnutyMoment_REAL > 0 THEN
//        P1_Srobovanie.STAV.M5_DosiahnutyMoment_REAL:= M5_DosiahnutyMoment_REAL/100;
//    ELSE
//        P1_Srobovanie.STAV.M5_DosiahnutyMoment_REAL:= 0.0;
//    END_IF

    M5_PrevodMomentu.AtlasAktualnyMoment:=P1_Srobovanie.PAR.M5_AtlasCopcoInputs[1];
    P1_Srobovanie.STAV.M5_DosiahnutyMoment_REAL:=M5_PrevodMomentu.AktualnyMoment;

    //Moment - Tolerancia MAX//
//    P1_Srobovanie.STAV.M5_Moment_ToleranciaMAX.0:= P1_Srobovanie.PAR.M5_AtlasCopcoInputs[3].24;
//    P1_Srobovanie.STAV.M5_Moment_ToleranciaMAX.1:= P1_Srobovanie.PAR.M5_AtlasCopcoInputs[3].25;
//    P1_Srobovanie.STAV.M5_Moment_ToleranciaMAX.2:= P1_Srobovanie.PAR.M5_AtlasCopcoInputs[3].26;
//    P1_Srobovanie.STAV.M5_Moment_ToleranciaMAX.3:= P1_Srobovanie.PAR.M5_AtlasCopcoInputs[3].27;
//    P1_Srobovanie.STAV.M5_Moment_ToleranciaMAX.4:= P1_Srobovanie.PAR.M5_AtlasCopcoInputs[3].28;
//    P1_Srobovanie.STAV.M5_Moment_ToleranciaMAX.5:= P1_Srobovanie.PAR.M5_AtlasCopcoInputs[3].29;
//    P1_Srobovanie.STAV.M5_Moment_ToleranciaMAX.6:= P1_Srobovanie.PAR.M5_AtlasCopcoInputs[3].30;
//    P1_Srobovanie.STAV.M5_Moment_ToleranciaMAX.7:= P1_Srobovanie.PAR.M5_AtlasCopcoInputs[3].31;
//    P1_Srobovanie.STAV.M5_Moment_ToleranciaMAX.8:= P1_Srobovanie.PAR.M5_AtlasCopcoInputs[3].16;
//    P1_Srobovanie.STAV.M5_Moment_ToleranciaMAX.9:= P1_Srobovanie.PAR.M5_AtlasCopcoInputs[3].17;
//    P1_Srobovanie.STAV.M5_Moment_ToleranciaMAX.10:= P1_Srobovanie.PAR.M5_AtlasCopcoInputs[3].18;
//    P1_Srobovanie.STAV.M5_Moment_ToleranciaMAX.11:= P1_Srobovanie.PAR.M5_AtlasCopcoInputs[3].19;
//    P1_Srobovanie.STAV.M5_Moment_ToleranciaMAX.12:= P1_Srobovanie.PAR.M5_AtlasCopcoInputs[3].20;
//    P1_Srobovanie.STAV.M5_Moment_ToleranciaMAX.13:= P1_Srobovanie.PAR.M5_AtlasCopcoInputs[3].21;
//    P1_Srobovanie.STAV.M5_Moment_ToleranciaMAX.14:= P1_Srobovanie.PAR.M5_AtlasCopcoInputs[3].22;
//    P1_Srobovanie.STAV.M5_Moment_ToleranciaMAX.15:= P1_Srobovanie.PAR.M5_AtlasCopcoInputs[3].23;
//    P1_Srobovanie.STAV.M5_Moment_ToleranciaMAX.16:= P1_Srobovanie.PAR.M5_AtlasCopcoInputs[3].8;
//    P1_Srobovanie.STAV.M5_Moment_ToleranciaMAX.17:= P1_Srobovanie.PAR.M5_AtlasCopcoInputs[3].9;
//    P1_Srobovanie.STAV.M5_Moment_ToleranciaMAX.18:= P1_Srobovanie.PAR.M5_AtlasCopcoInputs[3].10;
//    P1_Srobovanie.STAV.M5_Moment_ToleranciaMAX.19:= P1_Srobovanie.PAR.M5_AtlasCopcoInputs[3].11;
//    P1_Srobovanie.STAV.M5_Moment_ToleranciaMAX.20:= P1_Srobovanie.PAR.M5_AtlasCopcoInputs[3].12;
//    P1_Srobovanie.STAV.M5_Moment_ToleranciaMAX.21:= P1_Srobovanie.PAR.M5_AtlasCopcoInputs[3].13;
//    P1_Srobovanie.STAV.M5_Moment_ToleranciaMAX.22:= P1_Srobovanie.PAR.M5_AtlasCopcoInputs[3].14;
//    P1_Srobovanie.STAV.M5_Moment_ToleranciaMAX.23:= P1_Srobovanie.PAR.M5_AtlasCopcoInputs[3].15;
//    P1_Srobovanie.STAV.M5_Moment_ToleranciaMAX.24:= P1_Srobovanie.PAR.M5_AtlasCopcoInputs[3].0;
//    P1_Srobovanie.STAV.M5_Moment_ToleranciaMAX.25:= P1_Srobovanie.PAR.M5_AtlasCopcoInputs[3].1;
//    P1_Srobovanie.STAV.M5_Moment_ToleranciaMAX.26:= P1_Srobovanie.PAR.M5_AtlasCopcoInputs[3].2;
//    P1_Srobovanie.STAV.M5_Moment_ToleranciaMAX.27:= P1_Srobovanie.PAR.M5_AtlasCopcoInputs[3].3;
//    P1_Srobovanie.STAV.M5_Moment_ToleranciaMAX.28:= P1_Srobovanie.PAR.M5_AtlasCopcoInputs[3].4;
//    P1_Srobovanie.STAV.M5_Moment_ToleranciaMAX.29:= P1_Srobovanie.PAR.M5_AtlasCopcoInputs[3].5;
//    P1_Srobovanie.STAV.M5_Moment_ToleranciaMAX.30:= P1_Srobovanie.PAR.M5_AtlasCopcoInputs[3].6;
//    P1_Srobovanie.STAV.M5_Moment_ToleranciaMAX.31:= P1_Srobovanie.PAR.M5_AtlasCopcoInputs[3].7;
//    M5_Moment_ToleranciaMAX_REAL:= UDINT_TO_REAL(P1_Srobovanie.STAV.M5_Moment_ToleranciaMAX);
//    IF M5_Moment_ToleranciaMAX_REAL > 0 THEN
//        P1_Srobovanie.STAV.M5_Moment_ToleranciaMAX_REAL:= M5_Moment_ToleranciaMAX_REAL/100;
//    ELSE
//        P1_Srobovanie.STAV.M5_Moment_ToleranciaMAX_REAL:= 0.0;
    //    END_IF

    M5_PrevodMomentu.AtlasMaximalnaTolerancia:=P1_Srobovanie.PAR.M5_AtlasCopcoInputs[3];
    P1_Srobovanie.STAV.M5_Moment_ToleranciaMAX_REAL:=M5_PrevodMomentu.ToleranciaMAX;

    //Moment - Tolerancia MIN//
//    P1_Srobovanie.STAV.M5_Moment_ToleranciaMIN.0:= P1_Srobovanie.PAR.M5_AtlasCopcoInputs[4].24;
//    P1_Srobovanie.STAV.M5_Moment_ToleranciaMIN.1:= P1_Srobovanie.PAR.M5_AtlasCopcoInputs[4].25;
//    P1_Srobovanie.STAV.M5_Moment_ToleranciaMIN.2:= P1_Srobovanie.PAR.M5_AtlasCopcoInputs[4].26;
//    P1_Srobovanie.STAV.M5_Moment_ToleranciaMIN.3:= P1_Srobovanie.PAR.M5_AtlasCopcoInputs[4].27;
//    P1_Srobovanie.STAV.M5_Moment_ToleranciaMIN.4:= P1_Srobovanie.PAR.M5_AtlasCopcoInputs[4].28;
//    P1_Srobovanie.STAV.M5_Moment_ToleranciaMIN.5:= P1_Srobovanie.PAR.M5_AtlasCopcoInputs[4].29;
//    P1_Srobovanie.STAV.M5_Moment_ToleranciaMIN.6:= P1_Srobovanie.PAR.M5_AtlasCopcoInputs[4].30;
//    P1_Srobovanie.STAV.M5_Moment_ToleranciaMIN.7:= P1_Srobovanie.PAR.M5_AtlasCopcoInputs[4].31;
//    P1_Srobovanie.STAV.M5_Moment_ToleranciaMIN.8:= P1_Srobovanie.PAR.M5_AtlasCopcoInputs[4].16;
//    P1_Srobovanie.STAV.M5_Moment_ToleranciaMIN.9:= P1_Srobovanie.PAR.M5_AtlasCopcoInputs[4].17;
//    P1_Srobovanie.STAV.M5_Moment_ToleranciaMIN.10:= P1_Srobovanie.PAR.M5_AtlasCopcoInputs[4].18;
//    P1_Srobovanie.STAV.M5_Moment_ToleranciaMIN.11:= P1_Srobovanie.PAR.M5_AtlasCopcoInputs[4].19;
//    P1_Srobovanie.STAV.M5_Moment_ToleranciaMIN.12:= P1_Srobovanie.PAR.M5_AtlasCopcoInputs[4].20;
//    P1_Srobovanie.STAV.M5_Moment_ToleranciaMIN.13:= P1_Srobovanie.PAR.M5_AtlasCopcoInputs[4].21;
//    P1_Srobovanie.STAV.M5_Moment_ToleranciaMIN.14:= P1_Srobovanie.PAR.M5_AtlasCopcoInputs[4].22;
//    P1_Srobovanie.STAV.M5_Moment_ToleranciaMIN.15:= P1_Srobovanie.PAR.M5_AtlasCopcoInputs[4].23;
//    P1_Srobovanie.STAV.M5_Moment_ToleranciaMIN.16:= P1_Srobovanie.PAR.M5_AtlasCopcoInputs[4].8;
//    P1_Srobovanie.STAV.M5_Moment_ToleranciaMIN.17:= P1_Srobovanie.PAR.M5_AtlasCopcoInputs[4].9;
//    P1_Srobovanie.STAV.M5_Moment_ToleranciaMIN.18:= P1_Srobovanie.PAR.M5_AtlasCopcoInputs[4].10;
//    P1_Srobovanie.STAV.M5_Moment_ToleranciaMIN.19:= P1_Srobovanie.PAR.M5_AtlasCopcoInputs[4].11;
//    P1_Srobovanie.STAV.M5_Moment_ToleranciaMIN.20:= P1_Srobovanie.PAR.M5_AtlasCopcoInputs[4].12;
//    P1_Srobovanie.STAV.M5_Moment_ToleranciaMIN.21:= P1_Srobovanie.PAR.M5_AtlasCopcoInputs[4].13;
//    P1_Srobovanie.STAV.M5_Moment_ToleranciaMIN.22:= P1_Srobovanie.PAR.M5_AtlasCopcoInputs[4].14;
//    P1_Srobovanie.STAV.M5_Moment_ToleranciaMIN.23:= P1_Srobovanie.PAR.M5_AtlasCopcoInputs[4].15;
//    P1_Srobovanie.STAV.M5_Moment_ToleranciaMIN.24:= P1_Srobovanie.PAR.M5_AtlasCopcoInputs[4].0;
//    P1_Srobovanie.STAV.M5_Moment_ToleranciaMIN.25:= P1_Srobovanie.PAR.M5_AtlasCopcoInputs[4].1;
//    P1_Srobovanie.STAV.M5_Moment_ToleranciaMIN.26:= P1_Srobovanie.PAR.M5_AtlasCopcoInputs[4].2;
//    P1_Srobovanie.STAV.M5_Moment_ToleranciaMIN.27:= P1_Srobovanie.PAR.M5_AtlasCopcoInputs[4].3;
//    P1_Srobovanie.STAV.M5_Moment_ToleranciaMIN.28:= P1_Srobovanie.PAR.M5_AtlasCopcoInputs[4].4;
//    P1_Srobovanie.STAV.M5_Moment_ToleranciaMIN.29:= P1_Srobovanie.PAR.M5_AtlasCopcoInputs[4].5;
//    P1_Srobovanie.STAV.M5_Moment_ToleranciaMIN.30:= P1_Srobovanie.PAR.M5_AtlasCopcoInputs[4].6;
//    P1_Srobovanie.STAV.M5_Moment_ToleranciaMIN.31:= P1_Srobovanie.PAR.M5_AtlasCopcoInputs[4].7;
//    M5_Moment_ToleranciaMIN_REAL:= UDINT_TO_REAL(P1_Srobovanie.STAV.M5_Moment_ToleranciaMIN);
//    IF M5_Moment_ToleranciaMIN_REAL > 0 THEN
//        P1_Srobovanie.STAV.M5_Moment_ToleranciaMIN_REAL:= M5_Moment_ToleranciaMIN_REAL /100;
//    ELSE
//        P1_Srobovanie.STAV.M5_Moment_ToleranciaMIN_REAL:= 0.0;
    //    END_IF

    M5_PrevodMomentu.AtlasMinimalnaTolerancia:=P1_Srobovanie.PAR.M5_AtlasCopcoInputs[4];
    P1_Srobovanie.STAV.M5_Moment_ToleranciaMIN_REAL:=M5_PrevodMomentu.ToleranciaMIN;

    //Dosiahnutý úhol//
    P1_Srobovanie.STAV.M5_DosiahnutyUhol.0:= P1_Srobovanie.PAR.M5_AtlasCopcoInputs[0].24;
    P1_Srobovanie.STAV.M5_DosiahnutyUhol.1:= P1_Srobovanie.PAR.M5_AtlasCopcoInputs[0].25;
    P1_Srobovanie.STAV.M5_DosiahnutyUhol.2:= P1_Srobovanie.PAR.M5_AtlasCopcoInputs[0].26;
    P1_Srobovanie.STAV.M5_DosiahnutyUhol.3:= P1_Srobovanie.PAR.M5_AtlasCopcoInputs[0].27;
    P1_Srobovanie.STAV.M5_DosiahnutyUhol.4:= P1_Srobovanie.PAR.M5_AtlasCopcoInputs[0].28;
    P1_Srobovanie.STAV.M5_DosiahnutyUhol.5:= P1_Srobovanie.PAR.M5_AtlasCopcoInputs[0].29;
    P1_Srobovanie.STAV.M5_DosiahnutyUhol.6:= P1_Srobovanie.PAR.M5_AtlasCopcoInputs[0].30;
    P1_Srobovanie.STAV.M5_DosiahnutyUhol.7:= P1_Srobovanie.PAR.M5_AtlasCopcoInputs[0].31;
    P1_Srobovanie.STAV.M5_DosiahnutyUhol.8:= P1_Srobovanie.PAR.M5_AtlasCopcoInputs[0].16;
    P1_Srobovanie.STAV.M5_DosiahnutyUhol.9:= P1_Srobovanie.PAR.M5_AtlasCopcoInputs[0].17;
    P1_Srobovanie.STAV.M5_DosiahnutyUhol.10:= P1_Srobovanie.PAR.M5_AtlasCopcoInputs[0].18;
    P1_Srobovanie.STAV.M5_DosiahnutyUhol.11:= P1_Srobovanie.PAR.M5_AtlasCopcoInputs[0].19;
    P1_Srobovanie.STAV.M5_DosiahnutyUhol.12:= P1_Srobovanie.PAR.M5_AtlasCopcoInputs[0].20;
    P1_Srobovanie.STAV.M5_DosiahnutyUhol.13:= P1_Srobovanie.PAR.M5_AtlasCopcoInputs[0].21;
    P1_Srobovanie.STAV.M5_DosiahnutyUhol.14:= P1_Srobovanie.PAR.M5_AtlasCopcoInputs[0].22;
    P1_Srobovanie.STAV.M5_DosiahnutyUhol.15:= P1_Srobovanie.PAR.M5_AtlasCopcoInputs[0].23;

    //Uhol - Tolerancia MAX//
    P1_Srobovanie.STAV.M5_Uhol_ToleranciaMAX.0:= P1_Srobovanie.PAR.M5_AtlasCopcoInputs[2].8;
    P1_Srobovanie.STAV.M5_Uhol_ToleranciaMAX.1:= P1_Srobovanie.PAR.M5_AtlasCopcoInputs[2].9;
    P1_Srobovanie.STAV.M5_Uhol_ToleranciaMAX.2:= P1_Srobovanie.PAR.M5_AtlasCopcoInputs[2].10;
    P1_Srobovanie.STAV.M5_Uhol_ToleranciaMAX.3:= P1_Srobovanie.PAR.M5_AtlasCopcoInputs[2].11;
    P1_Srobovanie.STAV.M5_Uhol_ToleranciaMAX.4:= P1_Srobovanie.PAR.M5_AtlasCopcoInputs[2].12;
    P1_Srobovanie.STAV.M5_Uhol_ToleranciaMAX.5:= P1_Srobovanie.PAR.M5_AtlasCopcoInputs[2].13;
    P1_Srobovanie.STAV.M5_Uhol_ToleranciaMAX.6:= P1_Srobovanie.PAR.M5_AtlasCopcoInputs[2].14;
    P1_Srobovanie.STAV.M5_Uhol_ToleranciaMAX.7:= P1_Srobovanie.PAR.M5_AtlasCopcoInputs[2].15;
    P1_Srobovanie.STAV.M5_Uhol_ToleranciaMAX.8:= P1_Srobovanie.PAR.M5_AtlasCopcoInputs[2].0;
    P1_Srobovanie.STAV.M5_Uhol_ToleranciaMAX.9:= P1_Srobovanie.PAR.M5_AtlasCopcoInputs[2].1;
    P1_Srobovanie.STAV.M5_Uhol_ToleranciaMAX.10:= P1_Srobovanie.PAR.M5_AtlasCopcoInputs[2].2;
    P1_Srobovanie.STAV.M5_Uhol_ToleranciaMAX.11:= P1_Srobovanie.PAR.M5_AtlasCopcoInputs[2].3;
    P1_Srobovanie.STAV.M5_Uhol_ToleranciaMAX.12:= P1_Srobovanie.PAR.M5_AtlasCopcoInputs[2].4;
    P1_Srobovanie.STAV.M5_Uhol_ToleranciaMAX.13:= P1_Srobovanie.PAR.M5_AtlasCopcoInputs[2].5;
    P1_Srobovanie.STAV.M5_Uhol_ToleranciaMAX.14:= P1_Srobovanie.PAR.M5_AtlasCopcoInputs[2].6;
    P1_Srobovanie.STAV.M5_Uhol_ToleranciaMAX.15:= P1_Srobovanie.PAR.M5_AtlasCopcoInputs[2].7;

    //Uhol - Tolerancia MIN//
    P1_Srobovanie.STAV.M5_Uhol_ToleranciaMIN.0:= P1_Srobovanie.PAR.M5_AtlasCopcoInputs[2].24;
    P1_Srobovanie.STAV.M5_Uhol_ToleranciaMIN.1:= P1_Srobovanie.PAR.M5_AtlasCopcoInputs[2].25;
    P1_Srobovanie.STAV.M5_Uhol_ToleranciaMIN.2:= P1_Srobovanie.PAR.M5_AtlasCopcoInputs[2].26;
    P1_Srobovanie.STAV.M5_Uhol_ToleranciaMIN.3:= P1_Srobovanie.PAR.M5_AtlasCopcoInputs[2].27;
    P1_Srobovanie.STAV.M5_Uhol_ToleranciaMIN.4:= P1_Srobovanie.PAR.M5_AtlasCopcoInputs[2].28;
    P1_Srobovanie.STAV.M5_Uhol_ToleranciaMIN.5:= P1_Srobovanie.PAR.M5_AtlasCopcoInputs[2].29;
    P1_Srobovanie.STAV.M5_Uhol_ToleranciaMIN.6:= P1_Srobovanie.PAR.M5_AtlasCopcoInputs[2].30;
    P1_Srobovanie.STAV.M5_Uhol_ToleranciaMIN.7:= P1_Srobovanie.PAR.M5_AtlasCopcoInputs[2].31;
    P1_Srobovanie.STAV.M5_Uhol_ToleranciaMIN.8:= P1_Srobovanie.PAR.M5_AtlasCopcoInputs[2].16;
    P1_Srobovanie.STAV.M5_Uhol_ToleranciaMIN.9:= P1_Srobovanie.PAR.M5_AtlasCopcoInputs[2].17;
    P1_Srobovanie.STAV.M5_Uhol_ToleranciaMIN.10:= P1_Srobovanie.PAR.M5_AtlasCopcoInputs[2].18;
    P1_Srobovanie.STAV.M5_Uhol_ToleranciaMIN.11:= P1_Srobovanie.PAR.M5_AtlasCopcoInputs[2].19;
    P1_Srobovanie.STAV.M5_Uhol_ToleranciaMIN.12:= P1_Srobovanie.PAR.M5_AtlasCopcoInputs[2].20;
    P1_Srobovanie.STAV.M5_Uhol_ToleranciaMIN.13:= P1_Srobovanie.PAR.M5_AtlasCopcoInputs[2].21;
    P1_Srobovanie.STAV.M5_Uhol_ToleranciaMIN.14:= P1_Srobovanie.PAR.M5_AtlasCopcoInputs[2].22;
    P1_Srobovanie.STAV.M5_Uhol_ToleranciaMIN.15:= P1_Srobovanie.PAR.M5_AtlasCopcoInputs[2].23;

    //***************************************************************Skrutkovacka M4************************************************************************************//
    //Vstupy z AtlasCopco do PLC//
    P1_Srobovanie.Skrutkovacka_M4.Stav_VysledokPotvrdeny:= P1_Srobovanie.PAR.M4_AtlasCopcoInputs[0].0;
    P1_Srobovanie.Skrutkovacka_M4.Stav_EmergencyStop:= P1_Srobovanie.PAR.M4_AtlasCopcoInputs[0].1;
    P1_Srobovanie.Skrutkovacka_M4.Stav_READY_to_START:= P1_Srobovanie.PAR.M4_AtlasCopcoInputs[0].2;
    P1_Srobovanie.Skrutkovacka_M4.Stav_MANUAL:= P1_Srobovanie.PAR.M4_AtlasCopcoInputs[0].3;
    P1_Srobovanie.Skrutkovacka_M4.Stav_UtahovanieUkoncene:= P1_Srobovanie.PAR.M4_AtlasCopcoInputs[0].4;
    P1_Srobovanie.Skrutkovacka_M4.Stav_VysledokUtahovania_NG:= P1_Srobovanie.PAR.M4_AtlasCopcoInputs[0].5;
    P1_Srobovanie.Skrutkovacka_M4.Stav_VysledokUtahovania_OK:= P1_Srobovanie.PAR.M4_AtlasCopcoInputs[0].6;
    P1_Srobovanie.Skrutkovacka_M4.Stav_SmerOtacania_VPRED:= P1_Srobovanie.PAR.M4_AtlasCopcoInputs[0].7;
    P1_Srobovanie.Skrutkovacka_M4.Stav_BUSY:= P1_Srobovanie.PAR.M4_AtlasCopcoInputs[0].8;
    P1_Srobovanie.Skrutkovacka_M4.Stav_ControlerSwitch_ON:= P1_Srobovanie.PAR.M4_AtlasCopcoInputs[0].9;
    P1_Srobovanie.Skrutkovacka_M4.Stav_Station_READY:= P1_Srobovanie.PAR.M4_AtlasCopcoInputs[0].10;
    P1_Srobovanie.Skrutkovacka_M4.Stav_NastrojPripojeny:= P1_Srobovanie.PAR.M4_AtlasCopcoInputs[0].11;
    P1_Srobovanie.Skrutkovacka_M4.Stav_NastrojUtahuje:= P1_Srobovanie.PAR.M4_AtlasCopcoInputs[0].12;

    //Výstupy z PLC do AtlasCopco//
    P1_Srobovanie.PAR.M4_AllasCopcoOutputs[0].0:= P1_Srobovanie.Skrutkovacka_M4.RESET_Poruchy;
    P1_Srobovanie.PAR.M4_AllasCopcoOutputs[0].1:= P1_Srobovanie.Skrutkovacka_M4.RESET_Vysledkov;
    P1_Srobovanie.PAR.M4_AllasCopcoOutputs[0].2:= P1_Srobovanie.Skrutkovacka_M4.START_Skrutkovania;
    P1_Srobovanie.PAR.M4_AllasCopcoOutputs[0].3:= P1_Srobovanie.Skrutkovacka_M4.START_Utahovania;

    //Dosiahnutý moment//
//    P1_Srobovanie.STAV.M4_DosiahnutyMoment.0:= P1_Srobovanie.PAR.M4_AtlasCopcoInputs[1].24;
//    P1_Srobovanie.STAV.M4_DosiahnutyMoment.1:= P1_Srobovanie.PAR.M4_AtlasCopcoInputs[1].25;
//    P1_Srobovanie.STAV.M4_DosiahnutyMoment.2:= P1_Srobovanie.PAR.M4_AtlasCopcoInputs[1].26;
//    P1_Srobovanie.STAV.M4_DosiahnutyMoment.3:= P1_Srobovanie.PAR.M4_AtlasCopcoInputs[1].27;
//    P1_Srobovanie.STAV.M4_DosiahnutyMoment.4:= P1_Srobovanie.PAR.M4_AtlasCopcoInputs[1].28;
//    P1_Srobovanie.STAV.M4_DosiahnutyMoment.5:= P1_Srobovanie.PAR.M4_AtlasCopcoInputs[1].29;
//    P1_Srobovanie.STAV.M4_DosiahnutyMoment.6:= P1_Srobovanie.PAR.M4_AtlasCopcoInputs[1].30;
//    P1_Srobovanie.STAV.M4_DosiahnutyMoment.7:= P1_Srobovanie.PAR.M4_AtlasCopcoInputs[1].31;
//    P1_Srobovanie.STAV.M4_DosiahnutyMoment.8:= P1_Srobovanie.PAR.M4_AtlasCopcoInputs[1].16;
//    P1_Srobovanie.STAV.M4_DosiahnutyMoment.9:= P1_Srobovanie.PAR.M4_AtlasCopcoInputs[1].17;
//    P1_Srobovanie.STAV.M4_DosiahnutyMoment.10:= P1_Srobovanie.PAR.M4_AtlasCopcoInputs[1].18;
//    P1_Srobovanie.STAV.M4_DosiahnutyMoment.11:= P1_Srobovanie.PAR.M4_AtlasCopcoInputs[1].19;
//    P1_Srobovanie.STAV.M4_DosiahnutyMoment.12:= P1_Srobovanie.PAR.M4_AtlasCopcoInputs[1].20;
//    P1_Srobovanie.STAV.M4_DosiahnutyMoment.13:= P1_Srobovanie.PAR.M4_AtlasCopcoInputs[1].21;
//    P1_Srobovanie.STAV.M4_DosiahnutyMoment.14:= P1_Srobovanie.PAR.M4_AtlasCopcoInputs[1].22;
//    P1_Srobovanie.STAV.M4_DosiahnutyMoment.15:= P1_Srobovanie.PAR.M4_AtlasCopcoInputs[1].23;
//    P1_Srobovanie.STAV.M4_DosiahnutyMoment.16:= P1_Srobovanie.PAR.M4_AtlasCopcoInputs[1].8;
//    P1_Srobovanie.STAV.M4_DosiahnutyMoment.17:= P1_Srobovanie.PAR.M4_AtlasCopcoInputs[1].9;
//    P1_Srobovanie.STAV.M4_DosiahnutyMoment.18:= P1_Srobovanie.PAR.M4_AtlasCopcoInputs[1].10;
//    P1_Srobovanie.STAV.M4_DosiahnutyMoment.19:= P1_Srobovanie.PAR.M4_AtlasCopcoInputs[1].11;
//    P1_Srobovanie.STAV.M4_DosiahnutyMoment.20:= P1_Srobovanie.PAR.M4_AtlasCopcoInputs[1].12;
//    P1_Srobovanie.STAV.M4_DosiahnutyMoment.21:= P1_Srobovanie.PAR.M4_AtlasCopcoInputs[1].13;
//    P1_Srobovanie.STAV.M4_DosiahnutyMoment.22:= P1_Srobovanie.PAR.M4_AtlasCopcoInputs[1].14;
//    P1_Srobovanie.STAV.M4_DosiahnutyMoment.23:= P1_Srobovanie.PAR.M4_AtlasCopcoInputs[1].15;
//    P1_Srobovanie.STAV.M4_DosiahnutyMoment.24:= P1_Srobovanie.PAR.M4_AtlasCopcoInputs[1].0;
//    P1_Srobovanie.STAV.M4_DosiahnutyMoment.25:= P1_Srobovanie.PAR.M4_AtlasCopcoInputs[1].1;
//    P1_Srobovanie.STAV.M4_DosiahnutyMoment.26:= P1_Srobovanie.PAR.M4_AtlasCopcoInputs[1].2;
//    P1_Srobovanie.STAV.M4_DosiahnutyMoment.27:= P1_Srobovanie.PAR.M4_AtlasCopcoInputs[1].3;
//    P1_Srobovanie.STAV.M4_DosiahnutyMoment.28:= P1_Srobovanie.PAR.M4_AtlasCopcoInputs[1].4;
//    P1_Srobovanie.STAV.M4_DosiahnutyMoment.29:= P1_Srobovanie.PAR.M4_AtlasCopcoInputs[1].5;
//    P1_Srobovanie.STAV.M4_DosiahnutyMoment.30:= P1_Srobovanie.PAR.M4_AtlasCopcoInputs[1].6;
//    P1_Srobovanie.STAV.M4_DosiahnutyMoment.31:= P1_Srobovanie.PAR.M4_AtlasCopcoInputs[1].7;
//    M4_DosiahnutyMoment_REAL:= UDINT_TO_REAL(P1_Srobovanie.STAV.M4_DosiahnutyMoment);
//    IF M4_DosiahnutyMoment_REAL > 0 THEN
//        P1_Srobovanie.STAV.M4_DosiahnutyMoment_REAL:= (M4_DosiahnutyMoment_REAL*0.65)/42598;
//    ELSE
//        P1_Srobovanie.STAV.M4_DosiahnutyMoment_REAL:= 0.0;
//    END_IF

    M4_PrevodMomentu.AtlasAktualnyMoment:=P1_Srobovanie.PAR.M4_AtlasCopcoInputs[1];
    P1_Srobovanie.STAV.M4_DosiahnutyMoment_REAL:=M4_PrevodMomentu.AktualnyMoment;

    (*P1_Srobovanie.STAV.M4_DosiahnutyMoment_REAL:= M4_DosiahnutyMoment_REAL/100;*)

    //Moment - Tolerancia MAX//
//    P1_Srobovanie.STAV.M4_Moment_ToleranciaMAX.0:= P1_Srobovanie.PAR.M4_AtlasCopcoInputs[3].24;
    //    P1_Srobovanie.STAV.M4_Moment_ToleranciaMAX.1:= P1_Srobovanie.PAR.M4_AtlasCopcoInputs[3].25;
//    P1_Srobovanie.STAV.M4_Moment_ToleranciaMAX.2:= P1_Srobovanie.PAR.M4_AtlasCopcoInputs[3].26;
//    P1_Srobovanie.STAV.M4_Moment_ToleranciaMAX.3:= P1_Srobovanie.PAR.M4_AtlasCopcoInputs[3].27;
//    P1_Srobovanie.STAV.M4_Moment_ToleranciaMAX.4:= P1_Srobovanie.PAR.M4_AtlasCopcoInputs[3].28;
//    P1_Srobovanie.STAV.M4_Moment_ToleranciaMAX.5:= P1_Srobovanie.PAR.M4_AtlasCopcoInputs[3].29;
//    P1_Srobovanie.STAV.M4_Moment_ToleranciaMAX.6:= P1_Srobovanie.PAR.M4_AtlasCopcoInputs[3].30;
//    P1_Srobovanie.STAV.M4_Moment_ToleranciaMAX.7:= P1_Srobovanie.PAR.M4_AtlasCopcoInputs[3].31;
//    P1_Srobovanie.STAV.M4_Moment_ToleranciaMAX.8:= P1_Srobovanie.PAR.M4_AtlasCopcoInputs[3].16;
//    P1_Srobovanie.STAV.M4_Moment_ToleranciaMAX.9:= P1_Srobovanie.PAR.M4_AtlasCopcoInputs[3].17;
//    P1_Srobovanie.STAV.M4_Moment_ToleranciaMAX.10:= P1_Srobovanie.PAR.M4_AtlasCopcoInputs[3].18;
//    P1_Srobovanie.STAV.M4_Moment_ToleranciaMAX.11:= P1_Srobovanie.PAR.M4_AtlasCopcoInputs[3].19;
//    P1_Srobovanie.STAV.M4_Moment_ToleranciaMAX.12:= P1_Srobovanie.PAR.M4_AtlasCopcoInputs[3].20;
//    P1_Srobovanie.STAV.M4_Moment_ToleranciaMAX.13:= P1_Srobovanie.PAR.M4_AtlasCopcoInputs[3].21;
//    P1_Srobovanie.STAV.M4_Moment_ToleranciaMAX.14:= P1_Srobovanie.PAR.M4_AtlasCopcoInputs[3].22;
//    P1_Srobovanie.STAV.M4_Moment_ToleranciaMAX.15:= P1_Srobovanie.PAR.M4_AtlasCopcoInputs[3].23;
//    P1_Srobovanie.STAV.M4_Moment_ToleranciaMAX.16:= P1_Srobovanie.PAR.M4_AtlasCopcoInputs[3].8;
//    P1_Srobovanie.STAV.M4_Moment_ToleranciaMAX.17:= P1_Srobovanie.PAR.M4_AtlasCopcoInputs[3].9;
//    P1_Srobovanie.STAV.M4_Moment_ToleranciaMAX.18:= P1_Srobovanie.PAR.M4_AtlasCopcoInputs[3].10;
//    P1_Srobovanie.STAV.M4_Moment_ToleranciaMAX.19:= P1_Srobovanie.PAR.M4_AtlasCopcoInputs[3].11;
//    P1_Srobovanie.STAV.M4_Moment_ToleranciaMAX.20:= P1_Srobovanie.PAR.M4_AtlasCopcoInputs[3].12;
//    P1_Srobovanie.STAV.M4_Moment_ToleranciaMAX.21:= P1_Srobovanie.PAR.M4_AtlasCopcoInputs[3].13;
//    P1_Srobovanie.STAV.M4_Moment_ToleranciaMAX.22:= P1_Srobovanie.PAR.M4_AtlasCopcoInputs[3].14;
//    P1_Srobovanie.STAV.M4_Moment_ToleranciaMAX.23:= P1_Srobovanie.PAR.M4_AtlasCopcoInputs[3].15;
//    P1_Srobovanie.STAV.M4_Moment_ToleranciaMAX.24:= P1_Srobovanie.PAR.M4_AtlasCopcoInputs[3].0;
//    P1_Srobovanie.STAV.M4_Moment_ToleranciaMAX.25:= P1_Srobovanie.PAR.M4_AtlasCopcoInputs[3].1;
//    P1_Srobovanie.STAV.M4_Moment_ToleranciaMAX.26:= P1_Srobovanie.PAR.M4_AtlasCopcoInputs[3].2;
//    P1_Srobovanie.STAV.M4_Moment_ToleranciaMAX.27:= P1_Srobovanie.PAR.M4_AtlasCopcoInputs[3].3;
//    P1_Srobovanie.STAV.M4_Moment_ToleranciaMAX.28:= P1_Srobovanie.PAR.M4_AtlasCopcoInputs[3].4;
//    P1_Srobovanie.STAV.M4_Moment_ToleranciaMAX.29:= P1_Srobovanie.PAR.M4_AtlasCopcoInputs[3].5;
//    P1_Srobovanie.STAV.M4_Moment_ToleranciaMAX.30:= P1_Srobovanie.PAR.M4_AtlasCopcoInputs[3].6;
//    P1_Srobovanie.STAV.M4_Moment_ToleranciaMAX.31:= P1_Srobovanie.PAR.M4_AtlasCopcoInputs[3].7;
//    M4_Moment_ToleranciaMAX_REAL:= UDINT_TO_REAL(P1_Srobovanie.STAV.M4_Moment_ToleranciaMAX);
//    IF M4_Moment_ToleranciaMAX_REAL > 0 THEN
//        P1_Srobovanie.STAV.M4_Moment_ToleranciaMAX_REAL:= (M4_Moment_ToleranciaMAX_REAL*0.65)/42598;
//    ELSE
//        P1_Srobovanie.STAV.M4_Moment_ToleranciaMAX_REAL:= 0.0;
//    END_IF
    (*P1_Srobovanie.STAV.M4_Moment_ToleranciaMAX_REAL:= M4_Moment_ToleranciaMAX_REAL/100;*)

    M4_PrevodMomentu.AtlasMaximalnaTolerancia:=P1_Srobovanie.PAR.M4_AtlasCopcoInputs[3];
    P1_Srobovanie.STAV.M4_Moment_ToleranciaMAX_REAL:=M4_PrevodMomentu.ToleranciaMAX;

    //Moment - Tolerancia MIN//
//    P1_Srobovanie.STAV.M4_Moment_ToleranciaMIN.0:= P1_Srobovanie.PAR.M4_AtlasCopcoInputs[4].24;
//    P1_Srobovanie.STAV.M4_Moment_ToleranciaMIN.1:= P1_Srobovanie.PAR.M4_AtlasCopcoInputs[4].25;
//    P1_Srobovanie.STAV.M4_Moment_ToleranciaMIN.2:= P1_Srobovanie.PAR.M4_AtlasCopcoInputs[4].26;
//    P1_Srobovanie.STAV.M4_Moment_ToleranciaMIN.3:= P1_Srobovanie.PAR.M4_AtlasCopcoInputs[4].27;
//    P1_Srobovanie.STAV.M4_Moment_ToleranciaMIN.4:= P1_Srobovanie.PAR.M4_AtlasCopcoInputs[4].28;
//    P1_Srobovanie.STAV.M4_Moment_ToleranciaMIN.5:= P1_Srobovanie.PAR.M4_AtlasCopcoInputs[4].29;
//    P1_Srobovanie.STAV.M4_Moment_ToleranciaMIN.6:= P1_Srobovanie.PAR.M4_AtlasCopcoInputs[4].30;
//    P1_Srobovanie.STAV.M4_Moment_ToleranciaMIN.7:= P1_Srobovanie.PAR.M4_AtlasCopcoInputs[4].31;
//    P1_Srobovanie.STAV.M4_Moment_ToleranciaMIN.8:= P1_Srobovanie.PAR.M4_AtlasCopcoInputs[4].16;
//    P1_Srobovanie.STAV.M4_Moment_ToleranciaMIN.9:= P1_Srobovanie.PAR.M4_AtlasCopcoInputs[4].17;
//    P1_Srobovanie.STAV.M4_Moment_ToleranciaMIN.10:= P1_Srobovanie.PAR.M4_AtlasCopcoInputs[4].18;
//    P1_Srobovanie.STAV.M4_Moment_ToleranciaMIN.11:= P1_Srobovanie.PAR.M4_AtlasCopcoInputs[4].19;
//    P1_Srobovanie.STAV.M4_Moment_ToleranciaMIN.12:= P1_Srobovanie.PAR.M4_AtlasCopcoInputs[4].20;
//    P1_Srobovanie.STAV.M4_Moment_ToleranciaMIN.13:= P1_Srobovanie.PAR.M4_AtlasCopcoInputs[4].21;
//    P1_Srobovanie.STAV.M4_Moment_ToleranciaMIN.14:= P1_Srobovanie.PAR.M4_AtlasCopcoInputs[4].22;
//    P1_Srobovanie.STAV.M4_Moment_ToleranciaMIN.15:= P1_Srobovanie.PAR.M4_AtlasCopcoInputs[4].23;
//    P1_Srobovanie.STAV.M4_Moment_ToleranciaMIN.16:= P1_Srobovanie.PAR.M4_AtlasCopcoInputs[4].8;
//    P1_Srobovanie.STAV.M4_Moment_ToleranciaMIN.17:= P1_Srobovanie.PAR.M4_AtlasCopcoInputs[4].9;
//    P1_Srobovanie.STAV.M4_Moment_ToleranciaMIN.18:= P1_Srobovanie.PAR.M4_AtlasCopcoInputs[4].10;
//    P1_Srobovanie.STAV.M4_Moment_ToleranciaMIN.19:= P1_Srobovanie.PAR.M4_AtlasCopcoInputs[4].11;
//    P1_Srobovanie.STAV.M4_Moment_ToleranciaMIN.20:= P1_Srobovanie.PAR.M4_AtlasCopcoInputs[4].12;
//    P1_Srobovanie.STAV.M4_Moment_ToleranciaMIN.21:= P1_Srobovanie.PAR.M4_AtlasCopcoInputs[4].13;
//    P1_Srobovanie.STAV.M4_Moment_ToleranciaMIN.22:= P1_Srobovanie.PAR.M4_AtlasCopcoInputs[4].14;
//    P1_Srobovanie.STAV.M4_Moment_ToleranciaMIN.23:= P1_Srobovanie.PAR.M4_AtlasCopcoInputs[4].15;
//    P1_Srobovanie.STAV.M4_Moment_ToleranciaMIN.24:= P1_Srobovanie.PAR.M4_AtlasCopcoInputs[4].0;
//    P1_Srobovanie.STAV.M4_Moment_ToleranciaMIN.25:= P1_Srobovanie.PAR.M4_AtlasCopcoInputs[4].1;
//    P1_Srobovanie.STAV.M4_Moment_ToleranciaMIN.26:= P1_Srobovanie.PAR.M4_AtlasCopcoInputs[4].2;
//    P1_Srobovanie.STAV.M4_Moment_ToleranciaMIN.27:= P1_Srobovanie.PAR.M4_AtlasCopcoInputs[4].3;
//    P1_Srobovanie.STAV.M4_Moment_ToleranciaMIN.28:= P1_Srobovanie.PAR.M4_AtlasCopcoInputs[4].4;
//    P1_Srobovanie.STAV.M4_Moment_ToleranciaMIN.29:= P1_Srobovanie.PAR.M4_AtlasCopcoInputs[4].5;
//    P1_Srobovanie.STAV.M4_Moment_ToleranciaMIN.30:= P1_Srobovanie.PAR.M4_AtlasCopcoInputs[4].6;
//    P1_Srobovanie.STAV.M4_Moment_ToleranciaMIN.31:= P1_Srobovanie.PAR.M4_AtlasCopcoInputs[4].7;
//    M4_Moment_ToleranciaMIN_REAL:= UDINT_TO_REAL(P1_Srobovanie.STAV.M4_Moment_ToleranciaMIN);
//    IF M4_Moment_ToleranciaMIN_REAL > 0 THEN
//        P1_Srobovanie.STAV.M4_Moment_ToleranciaMIN_REAL:= (M4_Moment_ToleranciaMIN_REAL*0.65)/42598;
//    ELSE
//        P1_Srobovanie.STAV.M4_Moment_ToleranciaMIN_REAL:= 0.0;
//    END_IF
//
//
    (*P1_Srobovanie.STAV.M4_Moment_ToleranciaMIN_REAL:= M4_Moment_ToleranciaMIN_REAL /100;*)

    M4_PrevodMomentu.AtlasMinimalnaTolerancia:=P1_Srobovanie.PAR.M4_AtlasCopcoInputs[4];
    P1_Srobovanie.STAV.M4_Moment_ToleranciaMIN_REAL:=M4_PrevodMomentu.ToleranciaMIN;

    //Dosiahnutý úhol//
    P1_Srobovanie.STAV.M4_DosiahnutyUhol.0:= P1_Srobovanie.PAR.M4_AtlasCopcoInputs[0].24;
    P1_Srobovanie.STAV.M4_DosiahnutyUhol.1:= P1_Srobovanie.PAR.M4_AtlasCopcoInputs[0].25;
    P1_Srobovanie.STAV.M4_DosiahnutyUhol.2:= P1_Srobovanie.PAR.M4_AtlasCopcoInputs[0].26;
    P1_Srobovanie.STAV.M4_DosiahnutyUhol.3:= P1_Srobovanie.PAR.M4_AtlasCopcoInputs[0].27;
    P1_Srobovanie.STAV.M4_DosiahnutyUhol.4:= P1_Srobovanie.PAR.M4_AtlasCopcoInputs[0].28;
    P1_Srobovanie.STAV.M4_DosiahnutyUhol.5:= P1_Srobovanie.PAR.M4_AtlasCopcoInputs[0].29;
    P1_Srobovanie.STAV.M4_DosiahnutyUhol.6:= P1_Srobovanie.PAR.M4_AtlasCopcoInputs[0].30;
    P1_Srobovanie.STAV.M4_DosiahnutyUhol.7:= P1_Srobovanie.PAR.M4_AtlasCopcoInputs[0].31;
    P1_Srobovanie.STAV.M4_DosiahnutyUhol.8:= P1_Srobovanie.PAR.M4_AtlasCopcoInputs[0].16;
    P1_Srobovanie.STAV.M4_DosiahnutyUhol.9:= P1_Srobovanie.PAR.M4_AtlasCopcoInputs[0].17;
    P1_Srobovanie.STAV.M4_DosiahnutyUhol.10:= P1_Srobovanie.PAR.M4_AtlasCopcoInputs[0].18;
    P1_Srobovanie.STAV.M4_DosiahnutyUhol.11:= P1_Srobovanie.PAR.M4_AtlasCopcoInputs[0].19;
    P1_Srobovanie.STAV.M4_DosiahnutyUhol.12:= P1_Srobovanie.PAR.M4_AtlasCopcoInputs[0].20;
    P1_Srobovanie.STAV.M4_DosiahnutyUhol.13:= P1_Srobovanie.PAR.M4_AtlasCopcoInputs[0].21;
    P1_Srobovanie.STAV.M4_DosiahnutyUhol.14:= P1_Srobovanie.PAR.M4_AtlasCopcoInputs[0].22;
    P1_Srobovanie.STAV.M4_DosiahnutyUhol.15:= P1_Srobovanie.PAR.M4_AtlasCopcoInputs[0].23;

    //Uhol - Tolerancia MAX//
    P1_Srobovanie.STAV.M4_Uhol_ToleranciaMAX.0:= P1_Srobovanie.PAR.M4_AtlasCopcoInputs[2].8;
    P1_Srobovanie.STAV.M4_Uhol_ToleranciaMAX.1:= P1_Srobovanie.PAR.M4_AtlasCopcoInputs[2].9;
    P1_Srobovanie.STAV.M4_Uhol_ToleranciaMAX.2:= P1_Srobovanie.PAR.M4_AtlasCopcoInputs[2].10;
    P1_Srobovanie.STAV.M4_Uhol_ToleranciaMAX.3:= P1_Srobovanie.PAR.M4_AtlasCopcoInputs[2].11;
    P1_Srobovanie.STAV.M4_Uhol_ToleranciaMAX.4:= P1_Srobovanie.PAR.M4_AtlasCopcoInputs[2].12;
    P1_Srobovanie.STAV.M4_Uhol_ToleranciaMAX.5:= P1_Srobovanie.PAR.M4_AtlasCopcoInputs[2].13;
    P1_Srobovanie.STAV.M4_Uhol_ToleranciaMAX.6:= P1_Srobovanie.PAR.M4_AtlasCopcoInputs[2].14;
    P1_Srobovanie.STAV.M4_Uhol_ToleranciaMAX.7:= P1_Srobovanie.PAR.M4_AtlasCopcoInputs[2].15;
    P1_Srobovanie.STAV.M4_Uhol_ToleranciaMAX.8:= P1_Srobovanie.PAR.M4_AtlasCopcoInputs[2].0;
    P1_Srobovanie.STAV.M4_Uhol_ToleranciaMAX.9:= P1_Srobovanie.PAR.M4_AtlasCopcoInputs[2].1;
    P1_Srobovanie.STAV.M4_Uhol_ToleranciaMAX.10:= P1_Srobovanie.PAR.M4_AtlasCopcoInputs[2].2;
    P1_Srobovanie.STAV.M4_Uhol_ToleranciaMAX.11:= P1_Srobovanie.PAR.M4_AtlasCopcoInputs[2].3;
    P1_Srobovanie.STAV.M4_Uhol_ToleranciaMAX.12:= P1_Srobovanie.PAR.M4_AtlasCopcoInputs[2].4;
    P1_Srobovanie.STAV.M4_Uhol_ToleranciaMAX.13:= P1_Srobovanie.PAR.M4_AtlasCopcoInputs[2].5;
    P1_Srobovanie.STAV.M4_Uhol_ToleranciaMAX.14:= P1_Srobovanie.PAR.M4_AtlasCopcoInputs[2].6;
    P1_Srobovanie.STAV.M4_Uhol_ToleranciaMAX.15:= P1_Srobovanie.PAR.M4_AtlasCopcoInputs[2].7;

    //Uhol - Tolerancia MIN//
    P1_Srobovanie.STAV.M4_Uhol_ToleranciaMIN.0:= P1_Srobovanie.PAR.M4_AtlasCopcoInputs[2].24;
    P1_Srobovanie.STAV.M4_Uhol_ToleranciaMIN.1:= P1_Srobovanie.PAR.M4_AtlasCopcoInputs[2].25;
    P1_Srobovanie.STAV.M4_Uhol_ToleranciaMIN.2:= P1_Srobovanie.PAR.M4_AtlasCopcoInputs[2].26;
    P1_Srobovanie.STAV.M4_Uhol_ToleranciaMIN.3:= P1_Srobovanie.PAR.M4_AtlasCopcoInputs[2].27;
    P1_Srobovanie.STAV.M4_Uhol_ToleranciaMIN.4:= P1_Srobovanie.PAR.M4_AtlasCopcoInputs[2].28;
    P1_Srobovanie.STAV.M4_Uhol_ToleranciaMIN.5:= P1_Srobovanie.PAR.M4_AtlasCopcoInputs[2].29;
    P1_Srobovanie.STAV.M4_Uhol_ToleranciaMIN.6:= P1_Srobovanie.PAR.M4_AtlasCopcoInputs[2].30;
    P1_Srobovanie.STAV.M4_Uhol_ToleranciaMIN.7:= P1_Srobovanie.PAR.M4_AtlasCopcoInputs[2].31;
    P1_Srobovanie.STAV.M4_Uhol_ToleranciaMIN.8:= P1_Srobovanie.PAR.M4_AtlasCopcoInputs[2].16;
    P1_Srobovanie.STAV.M4_Uhol_ToleranciaMIN.9:= P1_Srobovanie.PAR.M4_AtlasCopcoInputs[2].17;
    P1_Srobovanie.STAV.M4_Uhol_ToleranciaMIN.10:= P1_Srobovanie.PAR.M4_AtlasCopcoInputs[2].18;
    P1_Srobovanie.STAV.M4_Uhol_ToleranciaMIN.11:= P1_Srobovanie.PAR.M4_AtlasCopcoInputs[2].19;
    P1_Srobovanie.STAV.M4_Uhol_ToleranciaMIN.12:= P1_Srobovanie.PAR.M4_AtlasCopcoInputs[2].20;
    P1_Srobovanie.STAV.M4_Uhol_ToleranciaMIN.13:= P1_Srobovanie.PAR.M4_AtlasCopcoInputs[2].21;
    P1_Srobovanie.STAV.M4_Uhol_ToleranciaMIN.14:= P1_Srobovanie.PAR.M4_AtlasCopcoInputs[2].22;
    P1_Srobovanie.STAV.M4_Uhol_ToleranciaMIN.15:= P1_Srobovanie.PAR.M4_AtlasCopcoInputs[2].23;

    //*********************************Skrutkovacka K30*******************************************************************************//
    //Vstupy z AtlasCopco do PLC//
    P1_Srobovanie.Skrutkovacka_K30.Stav_VysledokPotvrdeny:= P1_Srobovanie.PAR.K30_AtlasCopcoInputs[0].0;
    P1_Srobovanie.Skrutkovacka_K30.Stav_EmergencyStop:= P1_Srobovanie.PAR.K30_AtlasCopcoInputs[0].1;
    P1_Srobovanie.Skrutkovacka_K30.Stav_READY_to_START:= P1_Srobovanie.PAR.K30_AtlasCopcoInputs[0].2;
    P1_Srobovanie.Skrutkovacka_K30.Stav_MANUAL:= P1_Srobovanie.PAR.K30_AtlasCopcoInputs[0].3;
    P1_Srobovanie.Skrutkovacka_K30.Stav_UtahovanieUkoncene:= P1_Srobovanie.PAR.K30_AtlasCopcoInputs[0].4;
    P1_Srobovanie.Skrutkovacka_K30.Stav_VysledokUtahovania_NG:= P1_Srobovanie.PAR.K30_AtlasCopcoInputs[0].5;
    P1_Srobovanie.Skrutkovacka_K30.Stav_VysledokUtahovania_OK:= P1_Srobovanie.PAR.K30_AtlasCopcoInputs[0].6;
    P1_Srobovanie.Skrutkovacka_K30.Stav_SmerOtacania_VPRED:= P1_Srobovanie.PAR.K30_AtlasCopcoInputs[0].7;
    P1_Srobovanie.Skrutkovacka_K30.Stav_BUSY:= P1_Srobovanie.PAR.K30_AtlasCopcoInputs[0].8; //Další byte
    P1_Srobovanie.Skrutkovacka_K30.Stav_ControlerSwitch_ON:= P1_Srobovanie.PAR.K30_AtlasCopcoInputs[0].9;
    P1_Srobovanie.Skrutkovacka_K30.Stav_Station_READY:= P1_Srobovanie.PAR.K30_AtlasCopcoInputs[0].10;
    P1_Srobovanie.Skrutkovacka_K30.Stav_NastrojPripojeny:= P1_Srobovanie.PAR.K30_AtlasCopcoInputs[0].11;
    P1_Srobovanie.Skrutkovacka_K30.Stav_NastrojUtahuje:= P1_Srobovanie.PAR.K30_AtlasCopcoInputs[0].12;

    //Výstupy z PLC do AtlasCopco//
    P1_Srobovanie.PAR.K30_AllasCopcoOutputs[0].0:= P1_Srobovanie.Skrutkovacka_K30.RESET_Poruchy;
    P1_Srobovanie.PAR.K30_AllasCopcoOutputs[0].1:= P1_Srobovanie.Skrutkovacka_K30.RESET_Vysledkov;
    P1_Srobovanie.PAR.K30_AllasCopcoOutputs[0].2:= P1_Srobovanie.Skrutkovacka_K30.START_Skrutkovania;
    P1_Srobovanie.PAR.K30_AllasCopcoOutputs[0].3:= P1_Srobovanie.Skrutkovacka_K30.START_Utahovania;

    //Dosiahnutý moment//
//    P1_Srobovanie.STAV.K30_DosiahnutyMoment.0:= P1_Srobovanie.PAR.K30_AtlasCopcoInputs[1].24;
//    P1_Srobovanie.STAV.K30_DosiahnutyMoment.1:= P1_Srobovanie.PAR.K30_AtlasCopcoInputs[1].25;
//    P1_Srobovanie.STAV.K30_DosiahnutyMoment.2:= P1_Srobovanie.PAR.K30_AtlasCopcoInputs[1].26;
//    P1_Srobovanie.STAV.K30_DosiahnutyMoment.3:= P1_Srobovanie.PAR.K30_AtlasCopcoInputs[1].27;
//    P1_Srobovanie.STAV.K30_DosiahnutyMoment.4:= P1_Srobovanie.PAR.K30_AtlasCopcoInputs[1].28;
//    P1_Srobovanie.STAV.K30_DosiahnutyMoment.5:= P1_Srobovanie.PAR.K30_AtlasCopcoInputs[1].29;
//    P1_Srobovanie.STAV.K30_DosiahnutyMoment.6:= P1_Srobovanie.PAR.K30_AtlasCopcoInputs[1].30;
//    P1_Srobovanie.STAV.K30_DosiahnutyMoment.7:= P1_Srobovanie.PAR.K30_AtlasCopcoInputs[1].31;
//    P1_Srobovanie.STAV.K30_DosiahnutyMoment.8:= P1_Srobovanie.PAR.K30_AtlasCopcoInputs[1].16;
//    P1_Srobovanie.STAV.K30_DosiahnutyMoment.9:= P1_Srobovanie.PAR.K30_AtlasCopcoInputs[1].17;
//    P1_Srobovanie.STAV.K30_DosiahnutyMoment.10:= P1_Srobovanie.PAR.K30_AtlasCopcoInputs[1].18;
//    P1_Srobovanie.STAV.K30_DosiahnutyMoment.11:= P1_Srobovanie.PAR.K30_AtlasCopcoInputs[1].19;
//    P1_Srobovanie.STAV.K30_DosiahnutyMoment.12:= P1_Srobovanie.PAR.K30_AtlasCopcoInputs[1].20;
//    P1_Srobovanie.STAV.K30_DosiahnutyMoment.13:= P1_Srobovanie.PAR.K30_AtlasCopcoInputs[1].21;
//    P1_Srobovanie.STAV.K30_DosiahnutyMoment.14:= P1_Srobovanie.PAR.K30_AtlasCopcoInputs[1].22;
//    P1_Srobovanie.STAV.K30_DosiahnutyMoment.15:= P1_Srobovanie.PAR.K30_AtlasCopcoInputs[1].23;
//    P1_Srobovanie.STAV.K30_DosiahnutyMoment.16:= P1_Srobovanie.PAR.K30_AtlasCopcoInputs[1].8;
//    P1_Srobovanie.STAV.K30_DosiahnutyMoment.17:= P1_Srobovanie.PAR.K30_AtlasCopcoInputs[1].9;
//    P1_Srobovanie.STAV.K30_DosiahnutyMoment.18:= P1_Srobovanie.PAR.K30_AtlasCopcoInputs[1].10;
//    P1_Srobovanie.STAV.K30_DosiahnutyMoment.19:= P1_Srobovanie.PAR.K30_AtlasCopcoInputs[1].11;
//    P1_Srobovanie.STAV.K30_DosiahnutyMoment.20:= P1_Srobovanie.PAR.K30_AtlasCopcoInputs[1].12;
//    P1_Srobovanie.STAV.K30_DosiahnutyMoment.21:= P1_Srobovanie.PAR.K30_AtlasCopcoInputs[1].13;
//    P1_Srobovanie.STAV.K30_DosiahnutyMoment.22:= P1_Srobovanie.PAR.K30_AtlasCopcoInputs[1].14;
//    P1_Srobovanie.STAV.K30_DosiahnutyMoment.23:= P1_Srobovanie.PAR.K30_AtlasCopcoInputs[1].15;
//    P1_Srobovanie.STAV.K30_DosiahnutyMoment.24:= P1_Srobovanie.PAR.K30_AtlasCopcoInputs[1].0;
//    P1_Srobovanie.STAV.K30_DosiahnutyMoment.25:= P1_Srobovanie.PAR.K30_AtlasCopcoInputs[1].1;
//    P1_Srobovanie.STAV.K30_DosiahnutyMoment.26:= P1_Srobovanie.PAR.K30_AtlasCopcoInputs[1].2;
//    P1_Srobovanie.STAV.K30_DosiahnutyMoment.27:= P1_Srobovanie.PAR.K30_AtlasCopcoInputs[1].3;
//    P1_Srobovanie.STAV.K30_DosiahnutyMoment.28:= P1_Srobovanie.PAR.K30_AtlasCopcoInputs[1].4;
//    P1_Srobovanie.STAV.K30_DosiahnutyMoment.29:= P1_Srobovanie.PAR.K30_AtlasCopcoInputs[1].5;
//    P1_Srobovanie.STAV.K30_DosiahnutyMoment.30:= P1_Srobovanie.PAR.K30_AtlasCopcoInputs[1].6;
//    P1_Srobovanie.STAV.K30_DosiahnutyMoment.31:= P1_Srobovanie.PAR.K30_AtlasCopcoInputs[1].7;
//    K30_DosiahnutyMoment_REAL:= UDINT_TO_REAL(P1_Srobovanie.STAV.K30_DosiahnutyMoment);
//    IF K30_DosiahnutyMoment_REAL > 0 THEN
//        P1_Srobovanie.STAV.K30_DosiahnutyMoment_REAL:= K30_DosiahnutyMoment_REAL/100;
//    ELSE
//        P1_Srobovanie.STAV.K30_DosiahnutyMoment_REAL:= 0.0;
//    END_IF

    (*P1_Srobovanie.STAV.K30_DosiahnutyMoment_REAL:= (K30_DosiahnutyMoment_REAL*0.65)/42598;*)

    K30_PrevodMomentu.AtlasAktualnyMoment:=P1_Srobovanie.PAR.K30_AtlasCopcoInputs[1];
    P1_Srobovanie.STAV.K30_DosiahnutyMoment_REAL:=K30_PrevodMomentu.AktualnyMoment;

    //Moment - Tolerancia MAX//
//    P1_Srobovanie.STAV.K30_Moment_ToleranciaMAX.0:= P1_Srobovanie.PAR.K30_AtlasCopcoInputs[3].24;
//    P1_Srobovanie.STAV.K30_Moment_ToleranciaMAX.1:= P1_Srobovanie.PAR.K30_AtlasCopcoInputs[3].25;
//    P1_Srobovanie.STAV.K30_Moment_ToleranciaMAX.2:= P1_Srobovanie.PAR.K30_AtlasCopcoInputs[3].26;
//    P1_Srobovanie.STAV.K30_Moment_ToleranciaMAX.3:= P1_Srobovanie.PAR.K30_AtlasCopcoInputs[3].27;
//    P1_Srobovanie.STAV.K30_Moment_ToleranciaMAX.4:= P1_Srobovanie.PAR.K30_AtlasCopcoInputs[3].28;
//    P1_Srobovanie.STAV.K30_Moment_ToleranciaMAX.5:= P1_Srobovanie.PAR.K30_AtlasCopcoInputs[3].29;
//    P1_Srobovanie.STAV.K30_Moment_ToleranciaMAX.6:= P1_Srobovanie.PAR.K30_AtlasCopcoInputs[3].30;
//    P1_Srobovanie.STAV.K30_Moment_ToleranciaMAX.7:= P1_Srobovanie.PAR.K30_AtlasCopcoInputs[3].31;
//    P1_Srobovanie.STAV.K30_Moment_ToleranciaMAX.8:= P1_Srobovanie.PAR.K30_AtlasCopcoInputs[3].16;
//    P1_Srobovanie.STAV.K30_Moment_ToleranciaMAX.9:= P1_Srobovanie.PAR.K30_AtlasCopcoInputs[3].17;
//    P1_Srobovanie.STAV.K30_Moment_ToleranciaMAX.10:= P1_Srobovanie.PAR.K30_AtlasCopcoInputs[3].18;
//    P1_Srobovanie.STAV.K30_Moment_ToleranciaMAX.11:= P1_Srobovanie.PAR.K30_AtlasCopcoInputs[3].19;
//    P1_Srobovanie.STAV.K30_Moment_ToleranciaMAX.12:= P1_Srobovanie.PAR.K30_AtlasCopcoInputs[3].20;
//    P1_Srobovanie.STAV.K30_Moment_ToleranciaMAX.13:= P1_Srobovanie.PAR.K30_AtlasCopcoInputs[3].21;
//    P1_Srobovanie.STAV.K30_Moment_ToleranciaMAX.14:= P1_Srobovanie.PAR.K30_AtlasCopcoInputs[3].22;
//    P1_Srobovanie.STAV.K30_Moment_ToleranciaMAX.15:= P1_Srobovanie.PAR.K30_AtlasCopcoInputs[3].23;
//    P1_Srobovanie.STAV.K30_Moment_ToleranciaMAX.16:= P1_Srobovanie.PAR.K30_AtlasCopcoInputs[3].8;
//    P1_Srobovanie.STAV.K30_Moment_ToleranciaMAX.17:= P1_Srobovanie.PAR.K30_AtlasCopcoInputs[3].9;
//    P1_Srobovanie.STAV.K30_Moment_ToleranciaMAX.18:= P1_Srobovanie.PAR.K30_AtlasCopcoInputs[3].10;
//    P1_Srobovanie.STAV.K30_Moment_ToleranciaMAX.19:= P1_Srobovanie.PAR.K30_AtlasCopcoInputs[3].11;
//    P1_Srobovanie.STAV.K30_Moment_ToleranciaMAX.20:= P1_Srobovanie.PAR.K30_AtlasCopcoInputs[3].12;
//    P1_Srobovanie.STAV.K30_Moment_ToleranciaMAX.21:= P1_Srobovanie.PAR.K30_AtlasCopcoInputs[3].13;
//    P1_Srobovanie.STAV.K30_Moment_ToleranciaMAX.22:= P1_Srobovanie.PAR.K30_AtlasCopcoInputs[3].14;
//    P1_Srobovanie.STAV.K30_Moment_ToleranciaMAX.23:= P1_Srobovanie.PAR.K30_AtlasCopcoInputs[3].15;
//    P1_Srobovanie.STAV.K30_Moment_ToleranciaMAX.24:= P1_Srobovanie.PAR.K30_AtlasCopcoInputs[3].0;
//    P1_Srobovanie.STAV.K30_Moment_ToleranciaMAX.25:= P1_Srobovanie.PAR.K30_AtlasCopcoInputs[3].1;
//    P1_Srobovanie.STAV.K30_Moment_ToleranciaMAX.26:= P1_Srobovanie.PAR.K30_AtlasCopcoInputs[3].2;
//    P1_Srobovanie.STAV.K30_Moment_ToleranciaMAX.27:= P1_Srobovanie.PAR.K30_AtlasCopcoInputs[3].3;
//    P1_Srobovanie.STAV.K30_Moment_ToleranciaMAX.28:= P1_Srobovanie.PAR.K30_AtlasCopcoInputs[3].4;
//    P1_Srobovanie.STAV.K30_Moment_ToleranciaMAX.29:= P1_Srobovanie.PAR.K30_AtlasCopcoInputs[3].5;
//    P1_Srobovanie.STAV.K30_Moment_ToleranciaMAX.30:= P1_Srobovanie.PAR.K30_AtlasCopcoInputs[3].6;
//    P1_Srobovanie.STAV.K30_Moment_ToleranciaMAX.31:= P1_Srobovanie.PAR.K30_AtlasCopcoInputs[3].7;
//    K30_Moment_ToleranciaMAX_REAL:= UDINT_TO_REAL(P1_Srobovanie.STAV.K30_Moment_ToleranciaMAX);
//    IF K30_Moment_ToleranciaMAX_REAL > 0 THEN
//       P1_Srobovanie.STAV.K30_Moment_ToleranciaMAX_REAL:= K30_Moment_ToleranciaMAX_REAL/100;
//    ELSE
//        P1_Srobovanie.STAV.K30_Moment_ToleranciaMAX_REAL:= 0.0;
//    END_IF

    (*P1_Srobovanie.STAV.K30_Moment_ToleranciaMAX_REAL:= (K30_Moment_ToleranciaMAX_REAL*0.65)/42598;*)
    K30_PrevodMomentu.AtlasMaximalnaTolerancia:=P1_Srobovanie.PAR.K30_AtlasCopcoInputs[3];
    P1_Srobovanie.STAV.K30_Moment_ToleranciaMAX_REAL:=K30_PrevodMomentu.ToleranciaMAX;

    //Moment - Tolerancia MIN//
//    P1_Srobovanie.STAV.K30_Moment_ToleranciaMIN.0:= P1_Srobovanie.PAR.K30_AtlasCopcoInputs[4].24;
//    P1_Srobovanie.STAV.K30_Moment_ToleranciaMIN.1:= P1_Srobovanie.PAR.K30_AtlasCopcoInputs[4].25;
//    P1_Srobovanie.STAV.K30_Moment_ToleranciaMIN.2:= P1_Srobovanie.PAR.K30_AtlasCopcoInputs[4].26;
//    P1_Srobovanie.STAV.K30_Moment_ToleranciaMIN.3:= P1_Srobovanie.PAR.K30_AtlasCopcoInputs[4].27;
//    P1_Srobovanie.STAV.K30_Moment_ToleranciaMIN.4:= P1_Srobovanie.PAR.K30_AtlasCopcoInputs[4].28;
//    P1_Srobovanie.STAV.K30_Moment_ToleranciaMIN.5:= P1_Srobovanie.PAR.K30_AtlasCopcoInputs[4].29;
//    P1_Srobovanie.STAV.K30_Moment_ToleranciaMIN.6:= P1_Srobovanie.PAR.K30_AtlasCopcoInputs[4].30;
//    P1_Srobovanie.STAV.K30_Moment_ToleranciaMIN.7:= P1_Srobovanie.PAR.K30_AtlasCopcoInputs[4].31;
//    P1_Srobovanie.STAV.K30_Moment_ToleranciaMIN.8:= P1_Srobovanie.PAR.K30_AtlasCopcoInputs[4].16;
//    P1_Srobovanie.STAV.K30_Moment_ToleranciaMIN.9:= P1_Srobovanie.PAR.K30_AtlasCopcoInputs[4].17;
//    P1_Srobovanie.STAV.K30_Moment_ToleranciaMIN.10:= P1_Srobovanie.PAR.K30_AtlasCopcoInputs[4].18;
//    P1_Srobovanie.STAV.K30_Moment_ToleranciaMIN.11:= P1_Srobovanie.PAR.K30_AtlasCopcoInputs[4].19;
//    P1_Srobovanie.STAV.K30_Moment_ToleranciaMIN.12:= P1_Srobovanie.PAR.K30_AtlasCopcoInputs[4].20;
//    P1_Srobovanie.STAV.K30_Moment_ToleranciaMIN.13:= P1_Srobovanie.PAR.K30_AtlasCopcoInputs[4].21;
//    P1_Srobovanie.STAV.K30_Moment_ToleranciaMIN.14:= P1_Srobovanie.PAR.K30_AtlasCopcoInputs[4].22;
//    P1_Srobovanie.STAV.K30_Moment_ToleranciaMIN.15:= P1_Srobovanie.PAR.K30_AtlasCopcoInputs[4].23;
//    P1_Srobovanie.STAV.K30_Moment_ToleranciaMIN.16:= P1_Srobovanie.PAR.K30_AtlasCopcoInputs[4].8;
//    P1_Srobovanie.STAV.K30_Moment_ToleranciaMIN.17:= P1_Srobovanie.PAR.K30_AtlasCopcoInputs[4].9;
//    P1_Srobovanie.STAV.K30_Moment_ToleranciaMIN.18:= P1_Srobovanie.PAR.K30_AtlasCopcoInputs[4].10;
//    P1_Srobovanie.STAV.K30_Moment_ToleranciaMIN.19:= P1_Srobovanie.PAR.K30_AtlasCopcoInputs[4].11;
//    P1_Srobovanie.STAV.K30_Moment_ToleranciaMIN.20:= P1_Srobovanie.PAR.K30_AtlasCopcoInputs[4].12;
//    P1_Srobovanie.STAV.K30_Moment_ToleranciaMIN.21:= P1_Srobovanie.PAR.K30_AtlasCopcoInputs[4].13;
//    P1_Srobovanie.STAV.K30_Moment_ToleranciaMIN.22:= P1_Srobovanie.PAR.K30_AtlasCopcoInputs[4].14;
//    P1_Srobovanie.STAV.K30_Moment_ToleranciaMIN.23:= P1_Srobovanie.PAR.K30_AtlasCopcoInputs[4].15;
//    P1_Srobovanie.STAV.K30_Moment_ToleranciaMIN.24:= P1_Srobovanie.PAR.K30_AtlasCopcoInputs[4].0;
//    P1_Srobovanie.STAV.K30_Moment_ToleranciaMIN.25:= P1_Srobovanie.PAR.K30_AtlasCopcoInputs[4].1;
//    P1_Srobovanie.STAV.K30_Moment_ToleranciaMIN.26:= P1_Srobovanie.PAR.K30_AtlasCopcoInputs[4].2;
//    P1_Srobovanie.STAV.K30_Moment_ToleranciaMIN.27:= P1_Srobovanie.PAR.K30_AtlasCopcoInputs[4].3;
//    P1_Srobovanie.STAV.K30_Moment_ToleranciaMIN.28:= P1_Srobovanie.PAR.K30_AtlasCopcoInputs[4].4;
//    P1_Srobovanie.STAV.K30_Moment_ToleranciaMIN.29:= P1_Srobovanie.PAR.K30_AtlasCopcoInputs[4].5;
//    P1_Srobovanie.STAV.K30_Moment_ToleranciaMIN.30:= P1_Srobovanie.PAR.K30_AtlasCopcoInputs[4].6;
//    P1_Srobovanie.STAV.K30_Moment_ToleranciaMIN.31:= P1_Srobovanie.PAR.K30_AtlasCopcoInputs[4].7;
//    K30_Moment_ToleranciaMIN_REAL:= UDINT_TO_REAL(P1_Srobovanie.STAV.K30_Moment_ToleranciaMIN);
//    IF K30_Moment_ToleranciaMIN_REAL > 0 THEN
//        P1_Srobovanie.STAV.K30_Moment_ToleranciaMIN_REAL:= K30_Moment_ToleranciaMIN_REAL /100;
//    ELSE
//        P1_Srobovanie.STAV.K30_Moment_ToleranciaMIN_REAL:= 0.0;
//    END_IF

    (*P1_Srobovanie.STAV.K30_Moment_ToleranciaMIN_REAL:= (K30_Moment_ToleranciaMIN_REAL*0.65)/42598;*)
    K30_PrevodMomentu.AtlasMinimalnaTolerancia:=P1_Srobovanie.PAR.K30_AtlasCopcoInputs[4];
    P1_Srobovanie.STAV.K30_Moment_ToleranciaMIN_REAL:=K30_PrevodMomentu.ToleranciaMIN;

    //Dosiahnutý úhol//
    P1_Srobovanie.STAV.K30_DosiahnutyUhol.0:= P1_Srobovanie.PAR.K30_AtlasCopcoInputs[0].24;
    P1_Srobovanie.STAV.K30_DosiahnutyUhol.1:= P1_Srobovanie.PAR.K30_AtlasCopcoInputs[0].25;
    P1_Srobovanie.STAV.K30_DosiahnutyUhol.2:= P1_Srobovanie.PAR.K30_AtlasCopcoInputs[0].26;
    P1_Srobovanie.STAV.K30_DosiahnutyUhol.3:= P1_Srobovanie.PAR.K30_AtlasCopcoInputs[0].27;
    P1_Srobovanie.STAV.K30_DosiahnutyUhol.4:= P1_Srobovanie.PAR.K30_AtlasCopcoInputs[0].28;
    P1_Srobovanie.STAV.K30_DosiahnutyUhol.5:= P1_Srobovanie.PAR.K30_AtlasCopcoInputs[0].29;
    P1_Srobovanie.STAV.K30_DosiahnutyUhol.6:= P1_Srobovanie.PAR.K30_AtlasCopcoInputs[0].30;
    P1_Srobovanie.STAV.K30_DosiahnutyUhol.7:= P1_Srobovanie.PAR.K30_AtlasCopcoInputs[0].31;
    P1_Srobovanie.STAV.K30_DosiahnutyUhol.8:= P1_Srobovanie.PAR.K30_AtlasCopcoInputs[0].16;
    P1_Srobovanie.STAV.K30_DosiahnutyUhol.9:= P1_Srobovanie.PAR.K30_AtlasCopcoInputs[0].17;
    P1_Srobovanie.STAV.K30_DosiahnutyUhol.10:= P1_Srobovanie.PAR.K30_AtlasCopcoInputs[0].18;
    P1_Srobovanie.STAV.K30_DosiahnutyUhol.11:= P1_Srobovanie.PAR.K30_AtlasCopcoInputs[0].19;
    P1_Srobovanie.STAV.K30_DosiahnutyUhol.12:= P1_Srobovanie.PAR.K30_AtlasCopcoInputs[0].20;
    P1_Srobovanie.STAV.K30_DosiahnutyUhol.13:= P1_Srobovanie.PAR.K30_AtlasCopcoInputs[0].21;
    P1_Srobovanie.STAV.K30_DosiahnutyUhol.14:= P1_Srobovanie.PAR.K30_AtlasCopcoInputs[0].22;
    P1_Srobovanie.STAV.K30_DosiahnutyUhol.15:= P1_Srobovanie.PAR.K30_AtlasCopcoInputs[0].23;

    //Uhol - Tolerancia MAX//
    P1_Srobovanie.STAV.K30_Uhol_ToleranciaMAX.0:= P1_Srobovanie.PAR.K30_AtlasCopcoInputs[2].8;
    P1_Srobovanie.STAV.K30_Uhol_ToleranciaMAX.1:= P1_Srobovanie.PAR.K30_AtlasCopcoInputs[2].9;
    P1_Srobovanie.STAV.K30_Uhol_ToleranciaMAX.2:= P1_Srobovanie.PAR.K30_AtlasCopcoInputs[2].10;
    P1_Srobovanie.STAV.K30_Uhol_ToleranciaMAX.3:= P1_Srobovanie.PAR.K30_AtlasCopcoInputs[2].11;
    P1_Srobovanie.STAV.K30_Uhol_ToleranciaMAX.4:= P1_Srobovanie.PAR.K30_AtlasCopcoInputs[2].12;
    P1_Srobovanie.STAV.K30_Uhol_ToleranciaMAX.5:= P1_Srobovanie.PAR.K30_AtlasCopcoInputs[2].13;
    P1_Srobovanie.STAV.K30_Uhol_ToleranciaMAX.6:= P1_Srobovanie.PAR.K30_AtlasCopcoInputs[2].14;
    P1_Srobovanie.STAV.K30_Uhol_ToleranciaMAX.7:= P1_Srobovanie.PAR.K30_AtlasCopcoInputs[2].15;
    P1_Srobovanie.STAV.K30_Uhol_ToleranciaMAX.8:= P1_Srobovanie.PAR.K30_AtlasCopcoInputs[2].0;
    P1_Srobovanie.STAV.K30_Uhol_ToleranciaMAX.9:= P1_Srobovanie.PAR.K30_AtlasCopcoInputs[2].1;
    P1_Srobovanie.STAV.K30_Uhol_ToleranciaMAX.10:= P1_Srobovanie.PAR.K30_AtlasCopcoInputs[2].2;
    P1_Srobovanie.STAV.K30_Uhol_ToleranciaMAX.11:= P1_Srobovanie.PAR.K30_AtlasCopcoInputs[2].3;
    P1_Srobovanie.STAV.K30_Uhol_ToleranciaMAX.12:= P1_Srobovanie.PAR.K30_AtlasCopcoInputs[2].4;
    P1_Srobovanie.STAV.K30_Uhol_ToleranciaMAX.13:= P1_Srobovanie.PAR.K30_AtlasCopcoInputs[2].5;
    P1_Srobovanie.STAV.K30_Uhol_ToleranciaMAX.14:= P1_Srobovanie.PAR.K30_AtlasCopcoInputs[2].6;
    P1_Srobovanie.STAV.K30_Uhol_ToleranciaMAX.15:= P1_Srobovanie.PAR.K30_AtlasCopcoInputs[2].7;

    //Uhol - Tolerancia MIN//
    P1_Srobovanie.STAV.K30_Uhol_ToleranciaMIN.0:= P1_Srobovanie.PAR.K30_AtlasCopcoInputs[2].24;
    P1_Srobovanie.STAV.K30_Uhol_ToleranciaMIN.1:= P1_Srobovanie.PAR.K30_AtlasCopcoInputs[2].25;
    P1_Srobovanie.STAV.K30_Uhol_ToleranciaMIN.2:= P1_Srobovanie.PAR.K30_AtlasCopcoInputs[2].26;
    P1_Srobovanie.STAV.K30_Uhol_ToleranciaMIN.3:= P1_Srobovanie.PAR.K30_AtlasCopcoInputs[2].27;
    P1_Srobovanie.STAV.K30_Uhol_ToleranciaMIN.4:= P1_Srobovanie.PAR.K30_AtlasCopcoInputs[2].28;
    P1_Srobovanie.STAV.K30_Uhol_ToleranciaMIN.5:= P1_Srobovanie.PAR.K30_AtlasCopcoInputs[2].29;
    P1_Srobovanie.STAV.K30_Uhol_ToleranciaMIN.6:= P1_Srobovanie.PAR.K30_AtlasCopcoInputs[2].30;
    P1_Srobovanie.STAV.K30_Uhol_ToleranciaMIN.7:= P1_Srobovanie.PAR.K30_AtlasCopcoInputs[2].31;
    P1_Srobovanie.STAV.K30_Uhol_ToleranciaMIN.8:= P1_Srobovanie.PAR.K30_AtlasCopcoInputs[2].16;
    P1_Srobovanie.STAV.K30_Uhol_ToleranciaMIN.9:= P1_Srobovanie.PAR.K30_AtlasCopcoInputs[2].17;
    P1_Srobovanie.STAV.K30_Uhol_ToleranciaMIN.10:= P1_Srobovanie.PAR.K30_AtlasCopcoInputs[2].18;
    P1_Srobovanie.STAV.K30_Uhol_ToleranciaMIN.11:= P1_Srobovanie.PAR.K30_AtlasCopcoInputs[2].19;
    P1_Srobovanie.STAV.K30_Uhol_ToleranciaMIN.12:= P1_Srobovanie.PAR.K30_AtlasCopcoInputs[2].20;
    P1_Srobovanie.STAV.K30_Uhol_ToleranciaMIN.13:= P1_Srobovanie.PAR.K30_AtlasCopcoInputs[2].21;
    P1_Srobovanie.STAV.K30_Uhol_ToleranciaMIN.14:= P1_Srobovanie.PAR.K30_AtlasCopcoInputs[2].22;
    P1_Srobovanie.STAV.K30_Uhol_ToleranciaMIN.15:= P1_Srobovanie.PAR.K30_AtlasCopcoInputs[2].23;

END_ACTION
```

### Program Logical/Program/Pracovisko_1/P1_SkrutkovaciSet_K30 (IEC)
